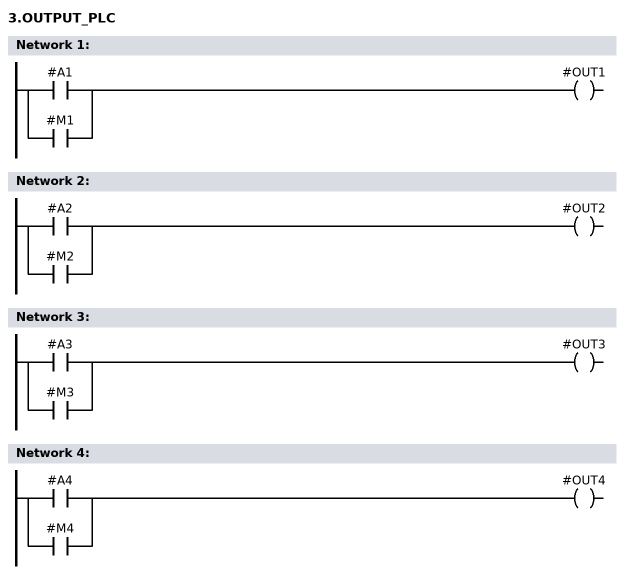
   RUNG wire#powerrail
      Contact( #A1 )
      wire#w1
      Coil( #OUT1 )
   END_RUNG
   RUNG wire#powerrail
      Contact( #M1 )
   END_RUNG wire#w1
   // the same network as SCL:
   #OUT1 := #A1 OR #M1;
END_REGION

REGION Network 2
   RUNG wire#powerrail
      Contact( #A2 )
      wire#w1
      Coil( #OUT2 )
   END_RUNG
   RUNG wire#powerrail
      Contact( #M2 )
   END_RUNG wire#w1
   // the same network as SCL:
   #OUT2 := #A2 OR #M2;
END_REGION

REGION Network 3
   RUNG wire#powerrail
      Contact( #A3 )
      wire#w1
      Coil( #OUT3 )
   END_RUNG
   RUNG wire#powerrail
      Contact( #M3 )
   END_RUNG wire#w1
   // the same network as SCL:
   #OUT3 := #A3 OR #M3;
END_REGION

REGION Network 4
   RUNG wire#powerrail
      Contact( #A4 )
      wire#w1
      Coil( #OUT4 )
   END_RUNG
   RUNG wire#powerrail
      Contact( #M4 )
   END_RUNG wire#w1
   // the same network as SCL:
   #OUT4 := #A4 OR #M4;
END_REGION
END_FUNCTION

FUNCTION_BLOCK "3.RUN_MODE"   // FB3, LAD
{ S7_Optimized_Access := 'TRUE' }
VERSION : 0.1
// stored: AutoNumber false, CodeModifiedDate 2025-08-27T17:11:43.2955348Z, CompileDate 2026-01-15T16:25:55.5692242Z, CreationDate 2026-01-15T16:22:49.8270549Z, DownloadWithoutReinit false, HandleErrorsWithinBlock false, InterfaceModifiedDate 2023-07-24T14:42:19.3789304Z, IsConsistent true, IsIECCheckEnabled false, IsKnowHowProtected false, IsRetainMemResEnabled false, IsWriteProtected false, LibraryConformanceStatus The object is library-conformant., MemoryReserve 100, ModifiedDate 2025-08-27T17:11:43.2955348Z, ParameterModified 2023-07-24T14:41:56.9787559Z, PLCSimAdvancedSupport false, SetENOAutomatically False, StructureModified 2023-07-24T14:42:19.3789304Z, UDAEnableTagReadback false
   VAR_INPUT
      NN_RUN : Bool;
      NN_STOP : Bool;
      SW_SIM : Bool;
      SW_MAN : Bool;
      SW_AUT : Bool;
   END_VAR
   VAR_OUTPUT
      RUN : Bool;
      SIM : Bool;
      MAN : Bool;
      AUT : Bool;
   END_VAR
   VAR
      TEMP1 : Bool;
      TEMP2 : Bool;
   END_VAR
BEGIN

REGION Network 1
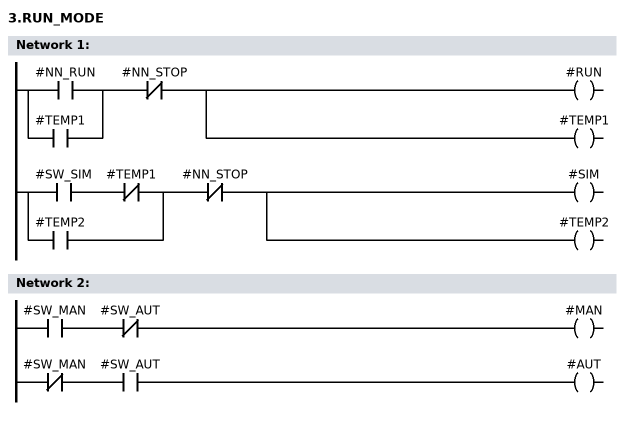
   RUNG wire#powerrail
      Contact( #NN_RUN )
      wire#w1
      I_Contact( #NN_STOP )
      wire#w2
      Coil( #RUN )
   END_RUNG
   RUNG wire#powerrail
      Contact( #TEMP1 )
   END_RUNG wire#w1
   RUNG wire#w2
      Coil( #TEMP1 )
   END_RUNG
   RUNG wire#powerrail
      Contact( #SW_SIM )
      I_Contact( #TEMP1 )
      wire#w3
      I_Contact( #NN_STOP )
      wire#w4
      Coil( #SIM )
   END_RUNG
   RUNG wire#powerrail
      Contact( #TEMP2 )
   END_RUNG wire#w3
   RUNG wire#w4
      Coil( #TEMP2 )
   END_RUNG
   // the same network as SCL:
   #RUN := (#NN_RUN OR #TEMP1) AND NOT #NN_STOP;
   #TEMP1 := #RUN;
   #SIM := ((#SW_SIM AND NOT #TEMP1) OR #TEMP2) AND NOT #NN_STOP;
   #TEMP2 := #SIM;
END_REGION

REGION Network 2
   RUNG wire#powerrail
      Contact( #SW_MAN )
      I_Contact( #SW_AUT )
      Coil( #MAN )
   END_RUNG
   RUNG wire#powerrail
      I_Contact( #SW_MAN )
      Contact( #SW_AUT )
      Coil( #AUT )
   END_RUNG
   // the same network as SCL:
   #MAN := #SW_MAN AND NOT #SW_AUT;
   #AUT := NOT #SW_MAN AND #SW_AUT;
END_REGION
END_FUNCTION_BLOCK

FUNCTION "4.CONVERT_VOLUME" : Void   // FC4, LAD
{ S7_Optimized_Access := 'TRUE' }
VERSION : 0.1
// stored: AutoNumber true, CodeModifiedDate 2025-08-27T17:08:03.467369Z, CompileDate 2026-01-15T16:25:55.7118746Z, CreationDate 2026-01-15T16:22:49.8270549Z, HandleErrorsWithinBlock false, InterfaceModifiedDate 2023-07-25T19:47:42.5745Z, IsConsistent true, IsIECCheckEnabled false, IsKnowHowProtected false, IsWriteProtected false, LibraryConformanceStatus The object is library-conformant., ModifiedDate 2025-08-27T17:08:03.467369Z, ParameterModified 2023-07-25T19:47:42.5745Z, PLCSimAdvancedSupport false, SetENOAutomatically False, StructureModified 2023-07-25T19:47:42.5745Z, UDAEnableTagReadback false
   VAR_INPUT
      SO_KHOI : Real;
      M3_MAX : Real;
   END_VAR
   VAR_OUTPUT
      SO_ME : Real;
      "M3/ME" : Real;
   END_VAR
   VAR_TEMP
      TEMP1 : Real;
      TEMP2 : Int;
      TEMP3 : Real;
   END_VAR
BEGIN

REGION Network 1
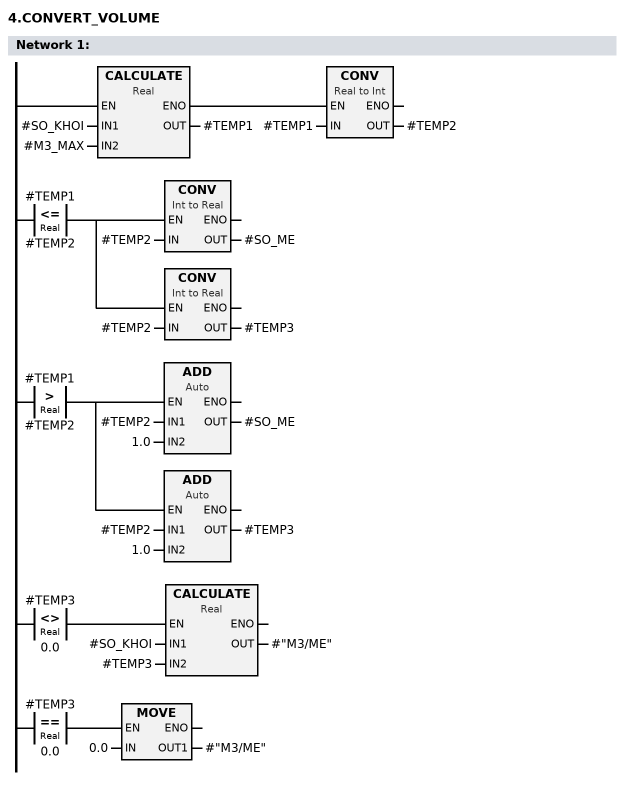
   RUNG wire#powerrail
      { S7_Templates := "SrcType := Real"; S7_Expression := "IN1/IN2" } Calculate(in1 := #SO_KHOI, in2 := #M3_MAX, out => #TEMP1)
      { S7_Templates := "[SrcType := Real, DestType := Int]" } Convert(in := #TEMP1, out => #TEMP2)
   END_RUNG
   RUNG wire#powerrail
      { S7_Templates := "SrcType := Real" } LE_Contact(in1 := #TEMP1, in2 := #TEMP2)
      wire#w1
      { S7_Templates := "[SrcType := Int, DestType := Real]" } Convert(in := #TEMP2, out => #SO_ME)
   END_RUNG
   RUNG wire#w1
      { S7_Templates := "[SrcType := Int, DestType := Real]" } Convert(in := #TEMP2, out => #TEMP3)
   END_RUNG
   RUNG wire#powerrail
      { S7_Templates := "SrcType := Real" } GT_Contact(in1 := #TEMP1, in2 := #TEMP2)
      wire#w2
      Add(in1 := #TEMP2, in2 := 1.0, out => #SO_ME)
   END_RUNG
   RUNG wire#w2
      Add(in1 := #TEMP2, in2 := 1.0, out => #TEMP3)
   END_RUNG
   RUNG wire#powerrail
      { S7_Templates := "SrcType := Real" } NE_Contact(in1 := #TEMP3, in2 := 0.0)
      { S7_Templates := "SrcType := Real"; S7_Expression := "IN1/IN2" } Calculate(in1 := #SO_KHOI, in2 := #TEMP3, out => #"M3/ME")
   END_RUNG
   RUNG wire#powerrail
      { S7_Templates := "SrcType := Real" } EQ_Contact(in1 := #TEMP3, in2 := 0.0)
      Move(in := 0.0, out1 => #"M3/ME")
   END_RUNG
   // the same network as SCL:
   #TEMP1 := #SO_KHOI/#M3_MAX;
   #TEMP2 := REAL_TO_INT(#TEMP1);
   IF #TEMP1 <= #TEMP2 THEN
       #SO_ME := INT_TO_REAL(#TEMP2);
       #TEMP3 := INT_TO_REAL(#TEMP2);
   END_IF;
   IF #TEMP1 > #TEMP2 THEN
       #SO_ME := #TEMP2 + 1.0;
       #TEMP3 := #TEMP2 + 1.0;
   END_IF;
   IF #TEMP3 <> 0.0 THEN #"M3/ME" := #SO_KHOI/#TEMP3; END_IF;
   IF #TEMP3 = 0.0 THEN #"M3/ME" := 0.0; END_IF;
END_REGION
END_FUNCTION

FUNCTION_BLOCK "5.ADDITIVES_PULE"   // FB5, LAD
{ S7_Optimized_Access := 'TRUE' }
VERSION : 0.1
// stored: AutoNumber false, CodeModifiedDate 2024-07-29T16:22:18.8856203Z, CompileDate 2026-01-15T16:25:55.5329987Z, CreationDate 2026-01-15T16:22:49.8270549Z, DownloadWithoutReinit false, HandleErrorsWithinBlock false, InterfaceModifiedDate 2024-07-29T16:20:48.5427985Z, IsConsistent true, IsIECCheckEnabled false, IsKnowHowProtected false, IsRetainMemResEnabled false, IsWriteProtected false, LibraryConformanceStatus The object is library-conformant., MemoryReserve 100, ModifiedDate 2024-07-29T16:22:18.8856203Z, ParameterModified 2024-07-29T16:20:48.5427985Z, PLCSimAdvancedSupport false, SetENOAutomatically False, StructureModified 2024-07-29T16:20:48.5427985Z, UDAEnableTagReadback false
   VAR_INPUT
      "Xung In" : DWord;
      Reset : Bool;
      "Set Tai" : Bool;
      "Khoi Luong Calib" : Real;
   END_VAR
   VAR_OUTPUT
      "Khoi Luong Out" : Real;
      "Xung Out" : Real;
   END_VAR
   VAR RETAIN
      "Xu In" : Real;
      "He So" : Real;
      "Xu Calib" : Real;
      "Kl Calib" : Real;
   END_VAR
   VAR
      M1 : Bool;
   END_VAR
   VAR_TEMP
      Conv : DInt;
   END_VAR
BEGIN

REGION Network 1
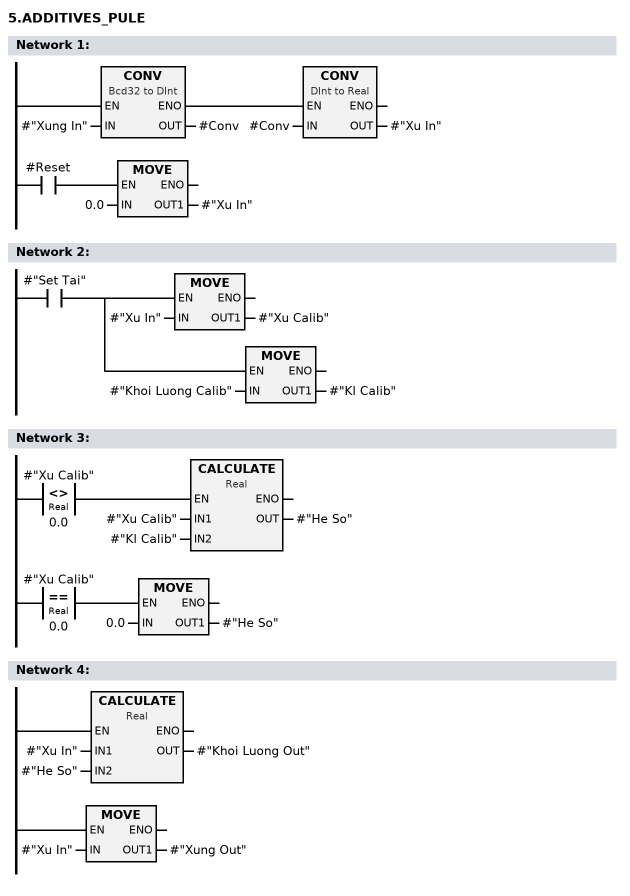
   RUNG wire#powerrail
      { S7_Templates := "[SrcType := Bcd32, DestType := DInt]" } Convert(in := #"Xung In", out => #Conv)
      { S7_Templates := "[SrcType := DInt, DestType := Real]" } Convert(in := #Conv, out => #"Xu In")
   END_RUNG
   RUNG wire#powerrail
      Contact( #Reset )
      Move(in := 0.0, out1 => #"Xu In")
   END_RUNG
   // the same network as SCL:
   #Conv := BCD32_TO_DINT(#"Xung In");
   #"Xu In" := DINT_TO_REAL(#Conv);
   IF #Reset THEN #"Xu In" := 0.0; END_IF;
END_REGION

REGION Network 2
   RUNG wire#powerrail
      Contact( #"Set Tai" )
      wire#w1
      Move(in := #"Xu In", out1 => #"Xu Calib")
   END_RUNG
   RUNG wire#w1
      Move(in := #"Khoi Luong Calib", out1 => #"Kl Calib")
   END_RUNG
   // the same network as SCL:
   IF #"Set Tai" THEN
       #"Xu Calib" := #"Xu In";
       #"Kl Calib" := #"Khoi Luong Calib";
   END_IF;
END_REGION

REGION Network 3
   RUNG wire#powerrail
      { S7_Templates := "SrcType := Real" } NE_Contact(in1 := #"Xu Calib", in2 := 0.0)
      { S7_Templates := "SrcType := Real"; S7_Expression := "IN2/IN1" } Calculate(in1 := #"Xu Calib", in2 := #"Kl Calib", out => #"He So")
   END_RUNG
   RUNG wire#powerrail
      { S7_Templates := "SrcType := Real" } EQ_Contact(in1 := #"Xu Calib", in2 := 0.0)
      Move(in := 0.0, out1 => #"He So")
   END_RUNG
   // the same network as SCL:
   IF #"Xu Calib" <> 0.0 THEN #"He So" := #"Kl Calib"/#"Xu Calib"; END_IF;
   IF #"Xu Calib" = 0.0 THEN #"He So" := 0.0; END_IF;
END_REGION

REGION Network 4
   RUNG wire#powerrail
      { S7_Templates := "SrcType := Real"; S7_Expression := "IN1*IN2" } Calculate(in1 := #"Xu In", in2 := #"He So", out => #"Khoi Luong Out")
   END_RUNG
   RUNG wire#powerrail
      Move(in := #"Xu In", out1 => #"Xung Out")
   END_RUNG
   // the same network as SCL:
   #"Khoi Luong Out" := #"Xu In"*#"He So";
   #"Xung Out" := #"Xu In";
END_REGION
END_FUNCTION_BLOCK

DATA_BLOCK "1.0 ANALOG_WAGG1"   // DB13
{ S7_Optimized_Access := 'TRUE' }
VERSION : 0.1
// stored: AutoNumber true, CodeModifiedDate 2026-01-15T16:25:52.6540779Z, CompileDate 2026-01-15T16:25:52.6593597Z, CreationDate 2026-01-15T16:22:49.8270549Z, DBAccessibleFromOPCUA true, DownloadWithoutReinit false, InstanceOfName 1.ANALOG_INPUT, InstanceOfNumber 1, InstanceOfType FB, InterfaceModifiedDate 2025-09-22T19:30:11.8403437Z, IsConsistent true, IsKnowHowProtected false, IsRetainMemResEnabled false, MemoryReserve 100, ModifiedDate 2026-01-15T16:25:52.6540779Z, ParameterModified 2025-08-30T17:31:01.4104373Z, StructureModified 2025-09-22T19:30:11.8403437Z, UDAEnableTagReadback false
"1.ANALOG_INPUT"
BEGIN
END_DATA_BLOCK

DATA_BLOCK "1.0 ANALOG_WAGG2"   // DB14
{ S7_Optimized_Access := 'TRUE' }
VERSION : 0.1
// stored: AutoNumber true, CodeModifiedDate 2026-01-15T16:25:52.3963656Z, CompileDate 2026-01-15T16:25:52.4020796Z, CreationDate 2026-01-15T16:22:49.8270549Z, DBAccessibleFromOPCUA true, DownloadWithoutReinit false, InstanceOfName 1.ANALOG_INPUT, InstanceOfNumber 1, InstanceOfType FB, InterfaceModifiedDate 2025-09-22T19:30:11.8403437Z, IsConsistent true, IsKnowHowProtected false, IsRetainMemResEnabled false, MemoryReserve 100, ModifiedDate 2026-01-15T16:25:52.3963656Z, ParameterModified 2025-08-30T17:31:01.4104373Z, StructureModified 2025-09-22T19:30:11.8403437Z, UDAEnableTagReadback false
"1.ANALOG_INPUT"
BEGIN
END_DATA_BLOCK

DATA_BLOCK "1.0 ANALOG_WAGG3"   // DB15
{ S7_Optimized_Access := 'TRUE' }
VERSION : 0.1
// stored: AutoNumber true, CodeModifiedDate 2026-01-15T16:25:52.7199099Z, CompileDate 2026-01-15T16:25:52.7268374Z, CreationDate 2026-01-15T16:22:49.8270549Z, DBAccessibleFromOPCUA true, DownloadWithoutReinit false, InstanceOfName 1.ANALOG_INPUT, InstanceOfNumber 1, InstanceOfType FB, InterfaceModifiedDate 2025-09-22T19:30:11.8403437Z, IsConsistent true, IsKnowHowProtected false, IsRetainMemResEnabled false, MemoryReserve 100, ModifiedDate 2026-01-15T16:25:52.7199099Z, ParameterModified 2025-08-30T17:31:01.4104373Z, StructureModified 2025-09-22T19:30:11.8403437Z, UDAEnableTagReadback false
"1.ANALOG_INPUT"
BEGIN
END_DATA_BLOCK

DATA_BLOCK "1.0 ANALOG_WAGG4"   // DB16
{ S7_Optimized_Access := 'TRUE' }
VERSION : 0.1
// stored: AutoNumber true, CodeModifiedDate 2026-01-15T16:25:52.7373182Z, CompileDate 2026-01-15T16:25:52.7414895Z, CreationDate 2026-01-15T16:22:49.8270549Z, DBAccessibleFromOPCUA true, DownloadWithoutReinit false, InstanceOfName 1.ANALOG_INPUT, InstanceOfNumber 1, InstanceOfType FB, InterfaceModifiedDate 2025-09-22T19:30:11.8403437Z, IsConsistent true, IsKnowHowProtected false, IsRetainMemResEnabled false, MemoryReserve 100, ModifiedDate 2026-01-15T16:25:52.7373182Z, ParameterModified 2025-08-30T17:31:01.4104373Z, StructureModified 2025-09-22T19:30:11.8403437Z, UDAEnableTagReadback false
"1.ANALOG_INPUT"
BEGIN
END_DATA_BLOCK

DATA_BLOCK "1.0 ANALOG_WAGG5"   // DB17
{ S7_Optimized_Access := 'TRUE' }
VERSION : 0.1
// stored: AutoNumber true, CodeModifiedDate 2026-01-15T16:25:52.7694615Z, CompileDate 2026-01-15T16:25:52.774821Z, CreationDate 2026-01-15T16:22:49.8270549Z, DBAccessibleFromOPCUA true, DownloadWithoutReinit false, InstanceOfName 1.ANALOG_INPUT, InstanceOfNumber 1, InstanceOfType FB, InterfaceModifiedDate 2025-09-22T19:30:11.8403437Z, IsConsistent true, IsKnowHowProtected false, IsRetainMemResEnabled false, MemoryReserve 100, ModifiedDate 2026-01-15T16:25:52.7694615Z, ParameterModified 2025-08-30T17:31:01.4104373Z, StructureModified 2025-09-22T19:30:11.8403437Z, UDAEnableTagReadback false
"1.ANALOG_INPUT"
BEGIN
END_DATA_BLOCK

DATA_BLOCK "1.0.ANALOG_WAG"   // DB100
{ S7_Optimized_Access := 'TRUE' }
VERSION : 0.1
// stored: AutoNumber false, CodeModifiedDate 2026-01-15T16:25:52.8141253Z, CompileDate 2026-01-15T16:25:52.8191872Z, CreationDate 2026-01-15T16:22:49.8270549Z, DBAccessibleFromOPCUA true, DownloadWithoutReinit false, InstanceOfName 1.ANALOG_INPUT, InstanceOfNumber 1, InstanceOfType FB, InterfaceModifiedDate 2025-09-22T19:30:11.8403437Z, IsConsistent true, IsKnowHowProtected false, IsRetainMemResEnabled false, MemoryReserve 100, ModifiedDate 2026-01-15T16:25:52.8141253Z, ParameterModified 2025-08-30T17:31:01.4104373Z, StructureModified 2025-09-22T19:30:11.8403437Z, UDAEnableTagReadback false
"1.ANALOG_INPUT"
BEGIN
END_DATA_BLOCK

DATA_BLOCK "1.0.ANALOG_WAP"   // DB102
{ S7_Optimized_Access := 'TRUE' }
VERSION : 0.1
// stored: AutoNumber false, CodeModifiedDate 2026-01-15T16:25:52.7536626Z, CompileDate 2026-01-15T16:25:52.7573094Z, CreationDate 2026-01-15T16:22:49.8270549Z, DBAccessibleFromOPCUA true, DownloadWithoutReinit false, InstanceOfName 1.ANALOG_INPUT, InstanceOfNumber 1, InstanceOfType FB, InterfaceModifiedDate 2025-09-22T19:30:11.8403437Z, IsConsistent true, IsKnowHowProtected false, IsRetainMemResEnabled false, MemoryReserve 100, ModifiedDate 2026-01-15T16:25:52.7536626Z, ParameterModified 2025-08-30T17:31:01.4104373Z, StructureModified 2025-09-22T19:30:11.8403437Z, UDAEnableTagReadback false
"1.ANALOG_INPUT"
BEGIN
END_DATA_BLOCK

DATA_BLOCK "1.0.ANALOG_WFD"   // DB101
{ S7_Optimized_Access := 'TRUE' }
VERSION : 0.1
// stored: AutoNumber false, CodeModifiedDate 2026-01-15T16:25:52.8468079Z, CompileDate 2026-01-15T16:25:52.8528873Z, CreationDate 2026-01-15T16:22:49.8270549Z, DBAccessibleFromOPCUA true, DownloadWithoutReinit false, InstanceOfName 1.ANALOG_INPUT, InstanceOfNumber 1, InstanceOfType FB, InterfaceModifiedDate 2025-09-22T19:30:11.8403437Z, IsConsistent true, IsKnowHowProtected false, IsRetainMemResEnabled false, MemoryReserve 100, ModifiedDate 2026-01-15T16:25:52.8468079Z, ParameterModified 2025-08-30T17:31:01.4104373Z, StructureModified 2025-09-22T19:30:11.8403437Z, UDAEnableTagReadback false
"1.ANALOG_INPUT"
BEGIN
END_DATA_BLOCK

DATA_BLOCK "1.0.ANALOG_WSBS"   // DB103
{ S7_Optimized_Access := 'TRUE' }
VERSION : 0.1
// stored: AutoNumber false, CodeModifiedDate 2026-01-15T16:25:52.4129937Z, CompileDate 2026-01-15T16:25:52.41757Z, CreationDate 2026-01-15T16:22:49.8270549Z, DBAccessibleFromOPCUA true, DownloadWithoutReinit false, InstanceOfName 1.ANALOG_INPUT, InstanceOfNumber 1, InstanceOfType FB, InterfaceModifiedDate 2025-09-22T19:30:11.8403437Z, IsConsistent true, IsKnowHowProtected false, IsRetainMemResEnabled false, MemoryReserve 100, ModifiedDate 2026-01-15T16:25:52.4129937Z, ParameterModified 2025-08-30T17:31:01.4104373Z, StructureModified 2025-09-22T19:30:11.8403437Z, UDAEnableTagReadback false
"1.ANALOG_INPUT"
BEGIN
END_DATA_BLOCK

DATA_BLOCK "1.1.ANALOG_TEMP_AG"   // DB107
{ S7_Optimized_Access := 'TRUE' }
VERSION : 0.1
// stored: AutoNumber false, CodeModifiedDate 2026-01-15T16:25:55.2427554Z, CompileDate 2026-01-15T16:25:55.2463904Z, CreationDate 2026-01-15T16:22:49.8270549Z, DBAccessibleFromOPCUA true, DownloadWithoutReinit false, InstanceOfName 1.ANALOG_INPUT, InstanceOfNumber 1, InstanceOfType FB, InterfaceModifiedDate 2025-09-22T19:30:11.8403437Z, IsConsistent true, IsKnowHowProtected false, IsRetainMemResEnabled false, MemoryReserve 100, ModifiedDate 2026-01-15T16:25:55.2427554Z, ParameterModified 2025-08-30T17:31:01.4104373Z, StructureModified 2025-09-22T19:30:11.8403437Z, UDAEnableTagReadback false
"1.ANALOG_INPUT"
BEGIN
END_DATA_BLOCK

DATA_BLOCK "1.1.ANALOG_TEMP_AP"   // DB106
{ S7_Optimized_Access := 'TRUE' }
VERSION : 0.1
// stored: AutoNumber false, CodeModifiedDate 2026-01-15T16:25:55.2265108Z, CompileDate 2026-01-15T16:25:55.2310383Z, CreationDate 2026-01-15T16:22:49.8270549Z, DBAccessibleFromOPCUA true, DownloadWithoutReinit false, InstanceOfName 1.ANALOG_INPUT, InstanceOfNumber 1, InstanceOfType FB, InterfaceModifiedDate 2025-09-22T19:30:11.8403437Z, IsConsistent true, IsKnowHowProtected false, IsRetainMemResEnabled false, MemoryReserve 100, ModifiedDate 2026-01-15T16:25:55.2265108Z, ParameterModified 2025-08-30T17:31:01.4104373Z, StructureModified 2025-09-22T19:30:11.8403437Z, UDAEnableTagReadback false
"1.ANALOG_INPUT"
BEGIN
END_DATA_BLOCK

DATA_BLOCK "1.1.ANALOG_TEMP_TL"   // DB104
{ S7_Optimized_Access := 'TRUE' }
VERSION : 0.1
// stored: AutoNumber false, CodeModifiedDate 2026-01-15T16:25:55.1844159Z, CompileDate 2026-01-15T16:25:55.1909886Z, CreationDate 2026-01-15T16:22:49.8270549Z, DBAccessibleFromOPCUA true, DownloadWithoutReinit false, InstanceOfName 1.ANALOG_INPUT, InstanceOfNumber 1, InstanceOfType FB, InterfaceModifiedDate 2025-09-22T19:30:11.8403437Z, IsConsistent true, IsKnowHowProtected false, IsRetainMemResEnabled false, MemoryReserve 100, ModifiedDate 2026-01-15T16:25:55.1844159Z, ParameterModified 2025-08-30T17:31:01.4104373Z, StructureModified 2025-09-22T19:30:11.8403437Z, UDAEnableTagReadback false
"1.ANALOG_INPUT"
BEGIN
END_DATA_BLOCK

DATA_BLOCK "1.1.ANALOG_TEMP_TS"   // DB105
{ S7_Optimized_Access := 'TRUE' }
VERSION : 0.1
// stored: AutoNumber false, CodeModifiedDate 2026-01-15T16:25:55.2062711Z, CompileDate 2026-01-15T16:25:55.2133319Z, CreationDate 2026-01-15T16:22:49.8270549Z, DBAccessibleFromOPCUA true, DownloadWithoutReinit false, InstanceOfName 1.ANALOG_INPUT, InstanceOfNumber 1, InstanceOfType FB, InterfaceModifiedDate 2025-09-22T19:30:11.8403437Z, IsConsistent true, IsKnowHowProtected false, IsRetainMemResEnabled false, MemoryReserve 100, ModifiedDate 2026-01-15T16:25:55.2062711Z, ParameterModified 2025-08-30T17:31:01.4104373Z, StructureModified 2025-09-22T19:30:11.8403437Z, UDAEnableTagReadback false
"1.ANALOG_INPUT"
BEGIN
END_DATA_BLOCK

DATA_BLOCK "10.0.RUNG_AGG1"   // DB1000
{ S7_Optimized_Access := 'TRUE' }
VERSION : 0.1
// stored: AutoNumber false, CodeModifiedDate 2026-01-15T16:25:55.7954208Z, CompileDate 2026-01-15T16:25:55.801975Z, CreationDate 2026-01-15T16:22:49.8270549Z, DBAccessibleFromOPCUA true, DownloadWithoutReinit false, InstanceOfName 10.TIMER_CLOCK, InstanceOfNumber 10, InstanceOfType FB, InterfaceModifiedDate 2023-08-14T08:08:19.3737097Z, IsConsistent true, IsKnowHowProtected false, IsRetainMemResEnabled false, MemoryReserve 100, ModifiedDate 2026-01-15T16:25:55.7954208Z, ParameterModified 2022-05-24T16:04:05.0982286Z, StructureModified 2023-08-14T08:08:19.3737097Z, UDAEnableTagReadback false
"10.TIMER_CLOCK"
BEGIN
END_DATA_BLOCK

DATA_BLOCK "10.1.RUNG_CE1"   // DB1006
{ S7_Optimized_Access := 'TRUE' }
VERSION : 0.1
// stored: AutoNumber false, CodeModifiedDate 2026-01-15T16:25:55.7775419Z, CompileDate 2026-01-15T16:25:55.7820883Z, CreationDate 2026-01-15T16:22:49.8270549Z, DBAccessibleFromOPCUA true, DownloadWithoutReinit false, InstanceOfName 10.TIMER_CLOCK, InstanceOfNumber 10, InstanceOfType FB, InterfaceModifiedDate 2023-08-14T08:08:19.3737097Z, IsConsistent true, IsKnowHowProtected false, IsRetainMemResEnabled false, MemoryReserve 100, ModifiedDate 2026-01-15T16:25:55.7775419Z, ParameterModified 2022-05-24T16:04:05.0982286Z, StructureModified 2023-08-14T08:08:19.3737097Z, UDAEnableTagReadback false
"10.TIMER_CLOCK"
BEGIN
END_DATA_BLOCK

DATA_BLOCK "10.3.SKSL_1"   // DB1009
{ S7_Optimized_Access := 'TRUE' }
VERSION : 0.1
// stored: AutoNumber false, CodeModifiedDate 2026-01-15T16:25:55.7623037Z, CompileDate 2026-01-15T16:25:55.7683704Z, CreationDate 2026-01-15T16:22:49.8270549Z, DBAccessibleFromOPCUA true, DownloadWithoutReinit false, InstanceOfName 10.TIMER_CLOCK, InstanceOfNumber 10, InstanceOfType FB, InterfaceModifiedDate 2023-08-14T08:08:19.3737097Z, IsConsistent true, IsKnowHowProtected false, IsRetainMemResEnabled false, MemoryReserve 100, ModifiedDate 2026-01-15T16:25:55.7623037Z, ParameterModified 2022-05-24T16:04:05.0982286Z, StructureModified 2023-08-14T08:08:19.3737097Z, UDAEnableTagReadback false
"10.TIMER_CLOCK"
BEGIN
END_DATA_BLOCK

DATA_BLOCK "2.0_NN0_0"   // DB200
{ S7_Optimized_Access := 'TRUE' }
VERSION : 0.1
// stored: AutoNumber false, CodeModifiedDate 2025-08-27T17:14:33.7093845Z, CompileDate 2026-01-15T16:25:52.803973Z, CreationDate 2026-01-15T16:22:49.8270549Z, DBAccessibleFromOPCUA true, DownloadWithoutReinit false, InstanceOfName 2.MANUAL_CONTROL, InstanceOfNumber 2, InstanceOfType FB, InterfaceModifiedDate 2025-08-27T17:14:33.2091456Z, IsConsistent true, IsKnowHowProtected false, IsRetainMemResEnabled false, MemoryReserve 100, ModifiedDate 2025-08-27T17:14:33.7093845Z, ParameterModified 2024-10-13T14:59:19.5830719Z, StructureModified 2025-08-27T17:14:33.2091456Z, UDAEnableTagReadback false
"2.MANUAL_CONTROL"
BEGIN
END_DATA_BLOCK

DATA_BLOCK "2.0_NN0_1"   // DB201
{ S7_Optimized_Access := 'TRUE' }
VERSION : 0.1
// stored: AutoNumber false, CodeModifiedDate 2025-08-27T17:14:33.6624193Z, CompileDate 2026-01-15T16:25:52.6174369Z, CreationDate 2026-01-15T16:22:49.8270549Z, DBAccessibleFromOPCUA true, DownloadWithoutReinit false, InstanceOfName 2.MANUAL_CONTROL, InstanceOfNumber 2, InstanceOfType FB, InterfaceModifiedDate 2025-08-27T17:14:33.2091456Z, IsConsistent true, IsKnowHowProtected false, IsRetainMemResEnabled false, MemoryReserve 100, ModifiedDate 2025-08-27T17:14:33.6624193Z, ParameterModified 2024-10-13T14:59:19.5830719Z, StructureModified 2025-08-27T17:14:33.2091456Z, UDAEnableTagReadback false
"2.MANUAL_CONTROL"
BEGIN
END_DATA_BLOCK

DATA_BLOCK "2.0_NN0_2"   // DB202
{ S7_Optimized_Access := 'TRUE' }
VERSION : 0.1
// stored: AutoNumber false, CodeModifiedDate 2025-08-27T17:14:33.8028627Z, CompileDate 2026-01-15T16:25:52.6287047Z, CreationDate 2026-01-15T16:22:49.8270549Z, DBAccessibleFromOPCUA true, DownloadWithoutReinit false, InstanceOfName 2.MANUAL_CONTROL, InstanceOfNumber 2, InstanceOfType FB, InterfaceModifiedDate 2025-08-27T17:14:33.2091456Z, IsConsistent true, IsKnowHowProtected false, IsRetainMemResEnabled false, MemoryReserve 100, ModifiedDate 2025-08-27T17:14:33.8028627Z, ParameterModified 2024-10-13T14:59:19.5830719Z, StructureModified 2025-08-27T17:14:33.2091456Z, UDAEnableTagReadback false
"2.MANUAL_CONTROL"
BEGIN
END_DATA_BLOCK

DATA_BLOCK "2.0_NN0_3"   // DB203
{ S7_Optimized_Access := 'TRUE' }
VERSION : 0.1
// stored: AutoNumber false, CodeModifiedDate 2025-08-27T17:14:33.7717804Z, CompileDate 2026-01-15T16:25:52.6419409Z, CreationDate 2026-01-15T16:22:49.8270549Z, DBAccessibleFromOPCUA true, DownloadWithoutReinit false, InstanceOfName 2.MANUAL_CONTROL, InstanceOfNumber 2, InstanceOfType FB, InterfaceModifiedDate 2025-08-27T17:14:33.2091456Z, IsConsistent true, IsKnowHowProtected false, IsRetainMemResEnabled false, MemoryReserve 100, ModifiedDate 2025-08-27T17:14:33.7717804Z, ParameterModified 2024-10-13T14:59:19.5830719Z, StructureModified 2025-08-27T17:14:33.2091456Z, UDAEnableTagReadback false
"2.MANUAL_CONTROL"
BEGIN
END_DATA_BLOCK

DATA_BLOCK "2.0_NN0_4"   // DB204
{ S7_Optimized_Access := 'TRUE' }
VERSION : 0.1
// stored: AutoNumber false, CodeModifiedDate 2025-08-27T17:14:33.7717798Z, CompileDate 2026-01-15T16:25:55.1732612Z, CreationDate 2026-01-15T16:22:49.8270549Z, DBAccessibleFromOPCUA true, DownloadWithoutReinit false, InstanceOfName 2.MANUAL_CONTROL, InstanceOfNumber 2, InstanceOfType FB, InterfaceModifiedDate 2025-08-27T17:14:33.2091456Z, IsConsistent true, IsKnowHowProtected false, IsRetainMemResEnabled false, MemoryReserve 100, ModifiedDate 2025-08-27T17:14:33.7717798Z, ParameterModified 2024-10-13T14:59:19.5830719Z, StructureModified 2025-08-27T17:14:33.2091456Z, UDAEnableTagReadback false
"2.MANUAL_CONTROL"
BEGIN
END_DATA_BLOCK

DATA_BLOCK "4.SIMULATION"   // DB400
{ S7_Optimized_Access := 'TRUE' }
VERSION : 0.1
// stored: AutoNumber false, CodeModifiedDate 2026-01-15T16:25:55.15091Z, CompileDate 2026-01-15T16:25:55.1580097Z, CreationDate 2026-01-15T16:22:49.8270549Z, DBAccessibleFromOPCUA true, DownloadWithoutReinit false, InstanceOfName 4.SIMULATION_DATA, InstanceOfNumber 4, InstanceOfType FB, InterfaceModifiedDate 2023-11-28T22:28:44.2264332Z, IsConsistent true, IsKnowHowProtected false, IsRetainMemResEnabled false, MemoryReserve 100, ModifiedDate 2026-01-15T16:25:55.15091Z, ParameterModified 2023-11-28T22:28:44.2264332Z, StructureModified 2023-11-28T22:28:44.2264332Z, UDAEnableTagReadback false
"4.SIMULATION_DATA"
BEGIN
END_DATA_BLOCK

DATA_BLOCK "6.1.WAGG1"   // DB601
{ S7_Optimized_Access := 'TRUE' }
VERSION : 0.1
// stored: AutoNumber false, CodeModifiedDate 2026-01-15T16:25:50.9109215Z, CompileDate 2026-01-15T16:25:50.9192936Z, CreationDate 2026-01-15T16:22:49.8270549Z, DBAccessibleFromOPCUA true, DownloadWithoutReinit false, InstanceOfName 6.WEIGHT_HANDLING, InstanceOfNumber 6, InstanceOfType FB, InterfaceModifiedDate 2023-12-29T17:39:18.5236469Z, IsConsistent true, IsKnowHowProtected false, IsRetainMemResEnabled false, MemoryReserve 100, ModifiedDate 2026-01-15T16:25:50.9109215Z, ParameterModified 2023-11-29T03:49:57.2782849Z, StructureModified 2023-12-29T17:39:18.5236469Z, UDAEnableTagReadback false
"6.WEIGHT_HANDLING"
BEGIN
END_DATA_BLOCK

DATA_BLOCK "6.1.W_IND_AGG1"   // DB19
{ S7_Optimized_Access := 'TRUE' }
VERSION : 0.1
// stored: AutoNumber true, CodeModifiedDate 2026-01-15T16:25:51.4257568Z, CompileDate 2026-01-15T16:25:51.429501Z, CreationDate 2026-01-15T16:22:49.8270549Z, DBAccessibleFromOPCUA true, DownloadWithoutReinit false, InstanceOfName 6.WEIGHT_HANDLING, InstanceOfNumber 6, InstanceOfType FB, InterfaceModifiedDate 2023-12-29T17:39:18.5236469Z, IsConsistent true, IsKnowHowProtected false, IsRetainMemResEnabled false, MemoryReserve 100, ModifiedDate 2026-01-15T16:25:51.4257568Z, ParameterModified 2023-11-29T03:49:57.2782849Z, StructureModified 2023-12-29T17:39:18.5236469Z, UDAEnableTagReadback false
"6.WEIGHT_HANDLING"
BEGIN
END_DATA_BLOCK

DATA_BLOCK "6.1.W_IND_AGG2"   // DB23
{ S7_Optimized_Access := 'TRUE' }
VERSION : 0.1
// stored: AutoNumber true, CodeModifiedDate 2026-01-15T16:25:52.0981926Z, CompileDate 2026-01-15T16:25:52.1042687Z, CreationDate 2026-01-15T16:22:49.8270549Z, DBAccessibleFromOPCUA true, DownloadWithoutReinit false, InstanceOfName 6.WEIGHT_HANDLING, InstanceOfNumber 6, InstanceOfType FB, InterfaceModifiedDate 2023-12-29T17:39:18.5236469Z, IsConsistent true, IsKnowHowProtected false, IsRetainMemResEnabled false, MemoryReserve 100, ModifiedDate 2026-01-15T16:25:52.0981926Z, ParameterModified 2023-11-29T03:49:57.2782849Z, StructureModified 2023-12-29T17:39:18.5236469Z, UDAEnableTagReadback false
"6.WEIGHT_HANDLING"
BEGIN
END_DATA_BLOCK

DATA_BLOCK "6.1.W_IND_AGG3"   // DB25
{ S7_Optimized_Access := 'TRUE' }
VERSION : 0.1
// stored: AutoNumber true, CodeModifiedDate 2026-01-15T16:25:52.1743928Z, CompileDate 2026-01-15T16:25:52.1820403Z, CreationDate 2026-01-15T16:22:49.8270549Z, DBAccessibleFromOPCUA true, DownloadWithoutReinit false, InstanceOfName 6.WEIGHT_HANDLING, InstanceOfNumber 6, InstanceOfType FB, InterfaceModifiedDate 2023-12-29T17:39:18.5236469Z, IsConsistent true, IsKnowHowProtected false, IsRetainMemResEnabled false, MemoryReserve 100, ModifiedDate 2026-01-15T16:25:52.1743928Z, ParameterModified 2023-11-29T03:49:57.2782849Z, StructureModified 2023-12-29T17:39:18.5236469Z, UDAEnableTagReadback false
"6.WEIGHT_HANDLING"
BEGIN
END_DATA_BLOCK

DATA_BLOCK "6.1.W_IND_AGG4"   // DB29
{ S7_Optimized_Access := 'TRUE' }
VERSION : 0.1
// stored: AutoNumber true, CodeModifiedDate 2026-01-15T16:25:52.0443037Z, CompileDate 2026-01-15T16:25:52.0495722Z, CreationDate 2026-01-15T16:22:49.8270549Z, DBAccessibleFromOPCUA true, DownloadWithoutReinit false, InstanceOfName 6.WEIGHT_HANDLING, InstanceOfNumber 6, InstanceOfType FB, InterfaceModifiedDate 2023-12-29T17:39:18.5236469Z, IsConsistent true, IsKnowHowProtected false, IsRetainMemResEnabled false, MemoryReserve 100, ModifiedDate 2026-01-15T16:25:52.0443037Z, ParameterModified 2023-11-29T03:49:57.2782849Z, StructureModified 2023-12-29T17:39:18.5236469Z, UDAEnableTagReadback false
"6.WEIGHT_HANDLING"
BEGIN
END_DATA_BLOCK

DATA_BLOCK "6.1.W_IND_AGG5"   // DB33
{ S7_Optimized_Access := 'TRUE' }
VERSION : 0.1
// stored: AutoNumber true, CodeModifiedDate 2026-01-15T16:25:51.9306777Z, CompileDate 2026-01-15T16:25:51.9357275Z, CreationDate 2026-01-15T16:22:49.8270549Z, DBAccessibleFromOPCUA true, DownloadWithoutReinit false, InstanceOfName 6.WEIGHT_HANDLING, InstanceOfNumber 6, InstanceOfType FB, InterfaceModifiedDate 2023-12-29T17:39:18.5236469Z, IsConsistent true, IsKnowHowProtected false, IsRetainMemResEnabled false, MemoryReserve 100, ModifiedDate 2026-01-15T16:25:51.9306777Z, ParameterModified 2023-11-29T03:49:57.2782849Z, StructureModified 2023-12-29T17:39:18.5236469Z, UDAEnableTagReadback false
"6.WEIGHT_HANDLING"
BEGIN
END_DATA_BLOCK

DATA_BLOCK "6.2.WCEM1"   // DB607
{ S7_Optimized_Access := 'TRUE' }
VERSION : 0.1
// stored: AutoNumber false, CodeModifiedDate 2026-01-15T16:25:51.2384683Z, CompileDate 2026-01-15T16:25:51.2440029Z, CreationDate 2026-01-15T16:22:49.8270549Z, DBAccessibleFromOPCUA true, DownloadWithoutReinit false, InstanceOfName 6.WEIGHT_HANDLING, InstanceOfNumber 6, InstanceOfType FB, InterfaceModifiedDate 2023-12-29T17:39:18.5236469Z, IsConsistent true, IsKnowHowProtected false, IsRetainMemResEnabled false, MemoryReserve 100, ModifiedDate 2026-01-15T16:25:51.2384683Z, ParameterModified 2023-11-29T03:49:57.2782849Z, StructureModified 2023-12-29T17:39:18.5236469Z, UDAEnableTagReadback false
"6.WEIGHT_HANDLING"
BEGIN
END_DATA_BLOCK

DATA_BLOCK "6.3.WWAT1"   // DB609
{ S7_Optimized_Access := 'TRUE' }
VERSION : 0.1
// stored: AutoNumber false, CodeModifiedDate 2026-01-15T16:25:51.1061526Z, CompileDate 2026-01-15T16:25:51.1117172Z, CreationDate 2026-01-15T16:22:49.8270549Z, DBAccessibleFromOPCUA true, DownloadWithoutReinit false, InstanceOfName 6.WEIGHT_HANDLING, InstanceOfNumber 6, InstanceOfType FB, InterfaceModifiedDate 2023-12-29T17:39:18.5236469Z, IsConsistent true, IsKnowHowProtected false, IsRetainMemResEnabled false, MemoryReserve 100, ModifiedDate 2026-01-15T16:25:51.1061526Z, ParameterModified 2023-11-29T03:49:57.2782849Z, StructureModified 2023-12-29T17:39:18.5236469Z, UDAEnableTagReadback false
"6.WEIGHT_HANDLING"
BEGIN
END_DATA_BLOCK

DATA_BLOCK "6.4.WADD1"   // DB611
{ S7_Optimized_Access := 'TRUE' }
VERSION : 0.1
// stored: AutoNumber false, CodeModifiedDate 2026-01-15T16:25:50.9806792Z, CompileDate 2026-01-15T16:25:50.9857091Z, CreationDate 2026-01-15T16:22:49.8270549Z, DBAccessibleFromOPCUA true, DownloadWithoutReinit false, InstanceOfName 6.WEIGHT_HANDLING, InstanceOfNumber 6, InstanceOfType FB, InterfaceModifiedDate 2023-12-29T17:39:18.5236469Z, IsConsistent true, IsKnowHowProtected false, IsRetainMemResEnabled false, MemoryReserve 100, ModifiedDate 2026-01-15T16:25:50.9806792Z, ParameterModified 2023-11-29T03:49:57.2782849Z, StructureModified 2023-12-29T17:39:18.5236469Z, UDAEnableTagReadback false
"6.WEIGHT_HANDLING"
BEGIN
END_DATA_BLOCK

DATA_BLOCK "7.1.AGG1"   // DB701
{ S7_Optimized_Access := 'TRUE' }
VERSION : 0.1
// stored: AutoNumber false, CodeModifiedDate 2026-01-15T16:25:50.9474767Z, CompileDate 2026-01-15T16:25:50.9530222Z, CreationDate 2026-01-15T16:22:49.8270549Z, DBAccessibleFromOPCUA true, DownloadWithoutReinit false, InstanceOfName 7.WEIGHT_PROCESS, InstanceOfNumber 7, InstanceOfType FB, InterfaceModifiedDate 2024-08-06T09:13:34.3012657Z, IsConsistent true, IsKnowHowProtected false, IsRetainMemResEnabled false, MemoryReserve 100, ModifiedDate 2026-01-15T16:25:50.9474767Z, ParameterModified 2024-08-06T08:53:48.4792275Z, StructureModified 2024-08-06T09:13:34.3012657Z, UDAEnableTagReadback false
"7.WEIGHT_PROCESS"
BEGIN
END_DATA_BLOCK

DATA_BLOCK "7.1.AGG2"   // DB702
{ S7_Optimized_Access := 'TRUE' }
VERSION : 0.1
// stored: AutoNumber false, CodeModifiedDate 2026-01-15T16:25:50.9657336Z, CompileDate 2026-01-15T16:25:50.9692801Z, CreationDate 2026-01-15T16:22:49.8270549Z, DBAccessibleFromOPCUA true, DownloadWithoutReinit false, InstanceOfName 7.WEIGHT_PROCESS, InstanceOfNumber 7, InstanceOfType FB, InterfaceModifiedDate 2024-08-06T09:13:34.3012657Z, IsConsistent true, IsKnowHowProtected false, IsRetainMemResEnabled false, MemoryReserve 100, ModifiedDate 2026-01-15T16:25:50.9657336Z, ParameterModified 2024-08-06T08:53:48.4792275Z, StructureModified 2024-08-06T09:13:34.3012657Z, UDAEnableTagReadback false
"7.WEIGHT_PROCESS"
BEGIN
END_DATA_BLOCK

DATA_BLOCK "7.1.AGG3"   // DB703
{ S7_Optimized_Access := 'TRUE' }
VERSION : 0.1
// stored: AutoNumber false, CodeModifiedDate 2026-01-15T16:25:51.0179497Z, CompileDate 2026-01-15T16:25:51.022606Z, CreationDate 2026-01-15T16:22:49.8270549Z, DBAccessibleFromOPCUA true, DownloadWithoutReinit false, InstanceOfName 7.WEIGHT_PROCESS, InstanceOfNumber 7, InstanceOfType FB, InterfaceModifiedDate 2024-08-06T09:13:34.3012657Z, IsConsistent true, IsKnowHowProtected false, IsRetainMemResEnabled false, MemoryReserve 100, ModifiedDate 2026-01-15T16:25:51.0179497Z, ParameterModified 2024-08-06T08:53:48.4792275Z, StructureModified 2024-08-06T09:13:34.3012657Z, UDAEnableTagReadback false
"7.WEIGHT_PROCESS"
BEGIN
END_DATA_BLOCK

DATA_BLOCK "7.1.AGG4"   // DB704
{ S7_Optimized_Access := 'TRUE' }
VERSION : 0.1
// stored: AutoNumber false, CodeModifiedDate 2026-01-15T16:25:51.0501858Z, CompileDate 2026-01-15T16:25:51.0579472Z, CreationDate 2026-01-15T16:22:49.8270549Z, DBAccessibleFromOPCUA true, DownloadWithoutReinit false, InstanceOfName 7.WEIGHT_PROCESS, InstanceOfNumber 7, InstanceOfType FB, InterfaceModifiedDate 2024-08-06T09:13:34.3012657Z, IsConsistent true, IsKnowHowProtected false, IsRetainMemResEnabled false, MemoryReserve 100, ModifiedDate 2026-01-15T16:25:51.0501858Z, ParameterModified 2024-08-06T08:53:48.4792275Z, StructureModified 2024-08-06T09:13:34.3012657Z, UDAEnableTagReadback false
"7.WEIGHT_PROCESS"
BEGIN
END_DATA_BLOCK

DATA_BLOCK "7.1.AGG5"   // DB705
{ S7_Optimized_Access := 'TRUE' }
VERSION : 0.1
// stored: AutoNumber false, CodeModifiedDate 2026-01-15T16:25:51.3893687Z, CompileDate 2026-01-15T16:25:51.396597Z, CreationDate 2026-01-15T16:22:49.8270549Z, DBAccessibleFromOPCUA true, DownloadWithoutReinit false, InstanceOfName 7.WEIGHT_PROCESS, InstanceOfNumber 7, InstanceOfType FB, InterfaceModifiedDate 2024-08-06T09:13:34.3012657Z, IsConsistent true, IsKnowHowProtected false, IsRetainMemResEnabled false, MemoryReserve 100, ModifiedDate 2026-01-15T16:25:51.3893687Z, ParameterModified 2024-08-06T08:53:48.4792275Z, StructureModified 2024-08-06T09:13:34.3012657Z, UDAEnableTagReadback false
"7.WEIGHT_PROCESS"
BEGIN
END_DATA_BLOCK

DATA_BLOCK "7.1.IND_AGG1"   // DB18
{ S7_Optimized_Access := 'TRUE' }
VERSION : 0.1
// stored: AutoNumber true, CodeModifiedDate 2026-01-15T16:25:52.372783Z, CompileDate 2026-01-15T16:25:52.3794201Z, CreationDate 2026-01-15T16:22:49.8270549Z, DBAccessibleFromOPCUA true, DownloadWithoutReinit false, InstanceOfName 7.WEIGHT_PROCESS, InstanceOfNumber 7, InstanceOfType FB, InterfaceModifiedDate 2024-08-06T09:13:34.3012657Z, IsConsistent true, IsKnowHowProtected false, IsRetainMemResEnabled false, MemoryReserve 100, ModifiedDate 2026-01-15T16:25:52.372783Z, ParameterModified 2024-08-06T08:53:48.4792275Z, StructureModified 2024-08-06T09:13:34.3012657Z, UDAEnableTagReadback false
"7.WEIGHT_PROCESS"
BEGIN
END_DATA_BLOCK

DATA_BLOCK "7.1.IND_AGG2"   // DB22
{ S7_Optimized_Access := 'TRUE' }
VERSION : 0.1
// stored: AutoNumber true, CodeModifiedDate 2026-01-15T16:25:52.2192426Z, CompileDate 2026-01-15T16:25:52.2239061Z, CreationDate 2026-01-15T16:22:49.8270549Z, DBAccessibleFromOPCUA true, DownloadWithoutReinit false, InstanceOfName 7.WEIGHT_PROCESS, InstanceOfNumber 7, InstanceOfType FB, InterfaceModifiedDate 2024-08-06T09:13:34.3012657Z, IsConsistent true, IsKnowHowProtected false, IsRetainMemResEnabled false, MemoryReserve 100, ModifiedDate 2026-01-15T16:25:52.2192426Z, ParameterModified 2024-08-06T08:53:48.4792275Z, StructureModified 2024-08-06T09:13:34.3012657Z, UDAEnableTagReadback false
"7.WEIGHT_PROCESS"
BEGIN
END_DATA_BLOCK

DATA_BLOCK "7.1.IND_AGG3"   // DB27
{ S7_Optimized_Access := 'TRUE' }
VERSION : 0.1
// stored: AutoNumber true, CodeModifiedDate 2026-01-15T16:25:52.0775696Z, CompileDate 2026-01-15T16:25:52.0841706Z, CreationDate 2026-01-15T16:22:49.8270549Z, DBAccessibleFromOPCUA true, DownloadWithoutReinit false, InstanceOfName 7.WEIGHT_PROCESS, InstanceOfNumber 7, InstanceOfType FB, InterfaceModifiedDate 2024-08-06T09:13:34.3012657Z, IsConsistent true, IsKnowHowProtected false, IsRetainMemResEnabled false, MemoryReserve 100, ModifiedDate 2026-01-15T16:25:52.0775696Z, ParameterModified 2024-08-06T08:53:48.4792275Z, StructureModified 2024-08-06T09:13:34.3012657Z, UDAEnableTagReadback false
"7.WEIGHT_PROCESS"
BEGIN
END_DATA_BLOCK

DATA_BLOCK "7.1.IND_AGG4"   // DB32
{ S7_Optimized_Access := 'TRUE' }
VERSION : 0.1
// stored: AutoNumber true, CodeModifiedDate 2026-01-15T16:25:52.1182917Z, CompileDate 2026-01-15T16:25:52.1243097Z, CreationDate 2026-01-15T16:22:49.8270549Z, DBAccessibleFromOPCUA true, DownloadWithoutReinit false, InstanceOfName 7.WEIGHT_PROCESS, InstanceOfNumber 7, InstanceOfType FB, InterfaceModifiedDate 2024-08-06T09:13:34.3012657Z, IsConsistent true, IsKnowHowProtected false, IsRetainMemResEnabled false, MemoryReserve 100, ModifiedDate 2026-01-15T16:25:52.1182917Z, ParameterModified 2024-08-06T08:53:48.4792275Z, StructureModified 2024-08-06T09:13:34.3012657Z, UDAEnableTagReadback false
"7.WEIGHT_PROCESS"
BEGIN
END_DATA_BLOCK

DATA_BLOCK "7.1.IND_AGG5"   // DB36
{ S7_Optimized_Access := 'TRUE' }
VERSION : 0.1
// stored: AutoNumber true, CodeModifiedDate 2026-01-15T16:25:52.0080123Z, CompileDate 2026-01-15T16:25:52.0131868Z, CreationDate 2026-01-15T16:22:49.8270549Z, DBAccessibleFromOPCUA true, DownloadWithoutReinit false, InstanceOfName 7.WEIGHT_PROCESS, InstanceOfNumber 7, InstanceOfType FB, InterfaceModifiedDate 2024-08-06T09:13:34.3012657Z, IsConsistent true, IsKnowHowProtected false, IsRetainMemResEnabled false, MemoryReserve 100, ModifiedDate 2026-01-15T16:25:52.0080123Z, ParameterModified 2024-08-06T08:53:48.4792275Z, StructureModified 2024-08-06T09:13:34.3012657Z, UDAEnableTagReadback false
"7.WEIGHT_PROCESS"
BEGIN
END_DATA_BLOCK

DATA_BLOCK "7.2.CE1"   // DB707
{ S7_Optimized_Access := 'TRUE' }
VERSION : 0.1
// stored: AutoNumber false, CodeModifiedDate 2026-01-15T16:25:50.7983554Z, CompileDate 2026-01-15T16:25:50.841758Z, CreationDate 2026-01-15T16:22:49.8270549Z, DBAccessibleFromOPCUA true, DownloadWithoutReinit false, InstanceOfName 7.WEIGHT_PROCESS, InstanceOfNumber 7, InstanceOfType FB, InterfaceModifiedDate 2024-08-06T09:13:34.3012657Z, IsConsistent true, IsKnowHowProtected false, IsRetainMemResEnabled false, MemoryReserve 100, ModifiedDate 2026-01-15T16:25:50.7983554Z, ParameterModified 2024-08-06T08:53:48.4792275Z, StructureModified 2024-08-06T09:13:34.3012657Z, UDAEnableTagReadback false
"7.WEIGHT_PROCESS"
BEGIN
END_DATA_BLOCK

DATA_BLOCK "7.3.WA1"   // DB712
{ S7_Optimized_Access := 'TRUE' }
VERSION : 0.1
// stored: AutoNumber false, CodeModifiedDate 2026-01-15T16:25:51.3687471Z, CompileDate 2026-01-15T16:25:51.3740828Z, CreationDate 2026-01-15T16:22:49.8270549Z, DBAccessibleFromOPCUA true, DownloadWithoutReinit false, InstanceOfName 7.WEIGHT_PROCESS, InstanceOfNumber 7, InstanceOfType FB, InterfaceModifiedDate 2024-08-06T09:13:34.3012657Z, IsConsistent true, IsKnowHowProtected false, IsRetainMemResEnabled false, MemoryReserve 100, ModifiedDate 2026-01-15T16:25:51.3687471Z, ParameterModified 2024-08-06T08:53:48.4792275Z, StructureModified 2024-08-06T09:13:34.3012657Z, UDAEnableTagReadback false
"7.WEIGHT_PROCESS"
BEGIN
END_DATA_BLOCK

DATA_BLOCK "7.4.ADD1"   // DB714
{ S7_Optimized_Access := 'TRUE' }
VERSION : 0.1
// stored: AutoNumber false, CodeModifiedDate 2026-01-15T16:25:50.880886Z, CompileDate 2026-01-15T16:25:50.8878267Z, CreationDate 2026-01-15T16:22:49.8270549Z, DBAccessibleFromOPCUA true, DownloadWithoutReinit false, InstanceOfName 7.WEIGHT_PROCESS, InstanceOfNumber 7, InstanceOfType FB, InterfaceModifiedDate 2024-08-06T09:13:34.3012657Z, IsConsistent true, IsKnowHowProtected false, IsRetainMemResEnabled false, MemoryReserve 100, ModifiedDate 2026-01-15T16:25:50.880886Z, ParameterModified 2024-08-06T08:53:48.4792275Z, StructureModified 2024-08-06T09:13:34.3012657Z, UDAEnableTagReadback false
"7.WEIGHT_PROCESS"
BEGIN
END_DATA_BLOCK

DATA_BLOCK "7.4.ADD2"   // DB715
{ S7_Optimized_Access := 'TRUE' }
VERSION : 0.1
// stored: AutoNumber true, CodeModifiedDate 2026-01-15T16:25:55.8171738Z, CompileDate 2026-01-15T16:25:55.8220055Z, CreationDate 2026-01-15T16:22:49.8270549Z, DBAccessibleFromOPCUA true, DownloadWithoutReinit false, InstanceOfName 7.WEIGHT_PROCESS, InstanceOfNumber 7, InstanceOfType FB, InterfaceModifiedDate 2024-08-06T09:13:34.3012657Z, IsConsistent true, IsKnowHowProtected false, IsRetainMemResEnabled false, MemoryReserve 100, ModifiedDate 2026-01-15T16:25:55.8171738Z, ParameterModified 2024-08-06T08:53:48.4792275Z, StructureModified 2024-08-06T09:13:34.3012657Z, UDAEnableTagReadback false
"7.WEIGHT_PROCESS"
BEGIN
END_DATA_BLOCK

DATA_BLOCK "7.4.ADD3"   // DB716
{ S7_Optimized_Access := 'TRUE' }
VERSION : 0.1
// stored: AutoNumber true, CodeModifiedDate 2026-01-15T16:25:55.4818033Z, CompileDate 2026-01-15T16:25:55.4875483Z, CreationDate 2026-01-15T16:22:49.8270549Z, DBAccessibleFromOPCUA true, DownloadWithoutReinit false, InstanceOfName 7.WEIGHT_PROCESS, InstanceOfNumber 7, InstanceOfType FB, InterfaceModifiedDate 2024-08-06T09:13:34.3012657Z, IsConsistent true, IsKnowHowProtected false, IsRetainMemResEnabled false, MemoryReserve 100, ModifiedDate 2026-01-15T16:25:55.4818033Z, ParameterModified 2024-08-06T08:53:48.4792275Z, StructureModified 2024-08-06T09:13:34.3012657Z, UDAEnableTagReadback false
"7.WEIGHT_PROCESS"
BEGIN
END_DATA_BLOCK

DATA_BLOCK "7.4.ADD4"   // DB717
{ S7_Optimized_Access := 'TRUE' }
VERSION : 0.1
// stored: AutoNumber true, CodeModifiedDate 2026-01-15T16:25:55.9772968Z, CompileDate 2026-01-15T16:25:55.9813329Z, CreationDate 2026-01-15T16:22:49.8270549Z, DBAccessibleFromOPCUA true, DownloadWithoutReinit false, InstanceOfName 7.WEIGHT_PROCESS, InstanceOfNumber 7, InstanceOfType FB, InterfaceModifiedDate 2024-08-06T09:13:34.3012657Z, IsConsistent true, IsKnowHowProtected false, IsRetainMemResEnabled false, MemoryReserve 100, ModifiedDate 2026-01-15T16:25:55.9772968Z, ParameterModified 2024-08-06T08:53:48.4792275Z, StructureModified 2024-08-06T09:13:34.3012657Z, UDAEnableTagReadback false
"7.WEIGHT_PROCESS"
BEGIN
END_DATA_BLOCK

DATA_BLOCK "7.4.ADD5"   // DB718
{ S7_Optimized_Access := 'TRUE' }
VERSION : 0.1
// stored: AutoNumber true, CodeModifiedDate 2026-01-15T16:25:55.9575787Z, CompileDate 2026-01-15T16:25:55.9634896Z, CreationDate 2026-01-15T16:22:49.8270549Z, DBAccessibleFromOPCUA true, DownloadWithoutReinit false, InstanceOfName 7.WEIGHT_PROCESS, InstanceOfNumber 7, InstanceOfType FB, InterfaceModifiedDate 2024-08-06T09:13:34.3012657Z, IsConsistent true, IsKnowHowProtected false, IsRetainMemResEnabled false, MemoryReserve 100, ModifiedDate 2026-01-15T16:25:55.9575787Z, ParameterModified 2024-08-06T08:53:48.4792275Z, StructureModified 2024-08-06T09:13:34.3012657Z, UDAEnableTagReadback false
"7.WEIGHT_PROCESS"
BEGIN
END_DATA_BLOCK

DATA_BLOCK "7.4.ADD6"   // DB719
{ S7_Optimized_Access := 'TRUE' }
VERSION : 0.1
// stored: AutoNumber true, CodeModifiedDate 2026-01-15T16:25:55.9362535Z, CompileDate 2026-01-15T16:25:55.9409287Z, CreationDate 2026-01-15T16:22:49.8270549Z, DBAccessibleFromOPCUA true, DownloadWithoutReinit false, InstanceOfName 7.WEIGHT_PROCESS, InstanceOfNumber 7, InstanceOfType FB, InterfaceModifiedDate 2024-08-06T09:13:34.3012657Z, IsConsistent true, IsKnowHowProtected false, IsRetainMemResEnabled false, MemoryReserve 100, ModifiedDate 2026-01-15T16:25:55.9362535Z, ParameterModified 2024-08-06T08:53:48.4792275Z, StructureModified 2024-08-06T09:13:34.3012657Z, UDAEnableTagReadback false
"7.WEIGHT_PROCESS"
BEGIN
END_DATA_BLOCK

DATA_BLOCK "9.1.DLC_AGG1"   // DB901
{ S7_Optimized_Access := 'TRUE' }
VERSION : 0.1
// stored: AutoNumber false, CodeModifiedDate 2026-01-15T16:25:50.9332093Z, CompileDate 2026-01-15T16:25:50.9377517Z, CreationDate 2026-01-15T16:22:49.8270549Z, DBAccessibleFromOPCUA true, DownloadWithoutReinit false, InstanceOfName 9.TIMER_DELAY, InstanceOfNumber 9, InstanceOfType FB, InterfaceModifiedDate 2022-05-24T16:36:11.1705081Z, IsConsistent true, IsKnowHowProtected false, IsRetainMemResEnabled false, MemoryReserve 100, ModifiedDate 2026-01-15T16:25:50.9332093Z, ParameterModified 2022-05-24T16:36:11.1705081Z, StructureModified 2022-05-24T16:36:11.1705081Z, UDAEnableTagReadback false
"9.TIMER_DELAY"
BEGIN
END_DATA_BLOCK

DATA_BLOCK "9.1.DLC_AGG2"   // DB902
{ S7_Optimized_Access := 'TRUE' }
VERSION : 0.1
// stored: AutoNumber false, CodeModifiedDate 2026-01-15T16:25:51.0711702Z, CompileDate 2026-01-15T16:25:51.0771226Z, CreationDate 2026-01-15T16:22:49.8270549Z, DBAccessibleFromOPCUA true, DownloadWithoutReinit false, InstanceOfName 9.TIMER_DELAY, InstanceOfNumber 9, InstanceOfType FB, InterfaceModifiedDate 2022-05-24T16:36:11.1705081Z, IsConsistent true, IsKnowHowProtected false, IsRetainMemResEnabled false, MemoryReserve 100, ModifiedDate 2026-01-15T16:25:51.0711702Z, ParameterModified 2022-05-24T16:36:11.1705081Z, StructureModified 2022-05-24T16:36:11.1705081Z, UDAEnableTagReadback false
"9.TIMER_DELAY"
BEGIN
END_DATA_BLOCK

DATA_BLOCK "9.1.DLC_AGG3"   // DB903
{ S7_Optimized_Access := 'TRUE' }
VERSION : 0.1
// stored: AutoNumber false, CodeModifiedDate 2026-01-15T16:25:50.9985443Z, CompileDate 2026-01-15T16:25:51.0044444Z, CreationDate 2026-01-15T16:22:49.8270549Z, DBAccessibleFromOPCUA true, DownloadWithoutReinit false, InstanceOfName 9.TIMER_DELAY, InstanceOfNumber 9, InstanceOfType FB, InterfaceModifiedDate 2022-05-24T16:36:11.1705081Z, IsConsistent true, IsKnowHowProtected false, IsRetainMemResEnabled false, MemoryReserve 100, ModifiedDate 2026-01-15T16:25:50.9985443Z, ParameterModified 2022-05-24T16:36:11.1705081Z, StructureModified 2022-05-24T16:36:11.1705081Z, UDAEnableTagReadback false
"9.TIMER_DELAY"
BEGIN
END_DATA_BLOCK

DATA_BLOCK "9.1.DLC_AGG4"   // DB904
{ S7_Optimized_Access := 'TRUE' }
VERSION : 0.1
// stored: AutoNumber false, CodeModifiedDate 2026-01-15T16:25:51.409636Z, CompileDate 2026-01-15T16:25:51.4146153Z, CreationDate 2026-01-15T16:22:49.8270549Z, DBAccessibleFromOPCUA true, DownloadWithoutReinit false, InstanceOfName 9.TIMER_DELAY, InstanceOfNumber 9, InstanceOfType FB, InterfaceModifiedDate 2022-05-24T16:36:11.1705081Z, IsConsistent true, IsKnowHowProtected false, IsRetainMemResEnabled false, MemoryReserve 100, ModifiedDate 2026-01-15T16:25:51.409636Z, ParameterModified 2022-05-24T16:36:11.1705081Z, StructureModified 2022-05-24T16:36:11.1705081Z, UDAEnableTagReadback false
"9.TIMER_DELAY"
BEGIN
END_DATA_BLOCK

DATA_BLOCK "9.1.DLC_AGG5"   // DB905
{ S7_Optimized_Access := 'TRUE' }
VERSION : 0.1
// stored: AutoNumber false, CodeModifiedDate 2026-01-15T16:25:51.1493744Z, CompileDate 2026-01-15T16:25:51.1554173Z, CreationDate 2026-01-15T16:22:49.8270549Z, DBAccessibleFromOPCUA true, DownloadWithoutReinit false, InstanceOfName 9.TIMER_DELAY, InstanceOfNumber 9, InstanceOfType FB, InterfaceModifiedDate 2022-05-24T16:36:11.1705081Z, IsConsistent true, IsKnowHowProtected false, IsRetainMemResEnabled false, MemoryReserve 100, ModifiedDate 2026-01-15T16:25:51.1493744Z, ParameterModified 2022-05-24T16:36:11.1705081Z, StructureModified 2022-05-24T16:36:11.1705081Z, UDAEnableTagReadback false
"9.TIMER_DELAY"
BEGIN
END_DATA_BLOCK

DATA_BLOCK "9.1.DLC_IND_AGG1"   // DB955
{ S7_Optimized_Access := 'TRUE' }
VERSION : 0.1
// stored: AutoNumber false, CodeModifiedDate 2026-01-15T16:25:52.3481914Z, CompileDate 2026-01-15T16:25:52.3557777Z, CreationDate 2026-01-15T16:22:49.8270549Z, DBAccessibleFromOPCUA true, DownloadWithoutReinit false, InstanceOfName 9.TIMER_DELAY, InstanceOfNumber 9, InstanceOfType FB, InterfaceModifiedDate 2022-05-24T16:36:11.1705081Z, IsConsistent true, IsKnowHowProtected false, IsRetainMemResEnabled false, MemoryReserve 100, ModifiedDate 2026-01-15T16:25:52.3481914Z, ParameterModified 2022-05-24T16:36:11.1705081Z, StructureModified 2022-05-24T16:36:11.1705081Z, UDAEnableTagReadback false
"9.TIMER_DELAY"
BEGIN
END_DATA_BLOCK

DATA_BLOCK "9.1.DLC_IND_AGG2"   // DB21
{ S7_Optimized_Access := 'TRUE' }
VERSION : 0.1
// stored: AutoNumber true, CodeModifiedDate 2026-01-15T16:25:51.3083868Z, CompileDate 2026-01-15T16:25:51.3114166Z, CreationDate 2026-01-15T16:22:49.8270549Z, DBAccessibleFromOPCUA true, DownloadWithoutReinit false, InstanceOfName 9.TIMER_DELAY, InstanceOfNumber 9, InstanceOfType FB, InterfaceModifiedDate 2022-05-24T16:36:11.1705081Z, IsConsistent true, IsKnowHowProtected false, IsRetainMemResEnabled false, MemoryReserve 100, ModifiedDate 2026-01-15T16:25:51.3083868Z, ParameterModified 2022-05-24T16:36:11.1705081Z, StructureModified 2022-05-24T16:36:11.1705081Z, UDAEnableTagReadback false
"9.TIMER_DELAY"
BEGIN
END_DATA_BLOCK

DATA_BLOCK "9.1.DLC_IND_AGG3"   // DB26
{ S7_Optimized_Access := 'TRUE' }
VERSION : 0.1
// stored: AutoNumber true, CodeModifiedDate 2026-01-15T16:25:51.2609627Z, CompileDate 2026-01-15T16:25:51.266563Z, CreationDate 2026-01-15T16:22:49.8270549Z, DBAccessibleFromOPCUA true, DownloadWithoutReinit false, InstanceOfName 9.TIMER_DELAY, InstanceOfNumber 9, InstanceOfType FB, InterfaceModifiedDate 2022-05-24T16:36:11.1705081Z, IsConsistent true, IsKnowHowProtected false, IsRetainMemResEnabled false, MemoryReserve 100, ModifiedDate 2026-01-15T16:25:51.2609627Z, ParameterModified 2022-05-24T16:36:11.1705081Z, StructureModified 2022-05-24T16:36:11.1705081Z, UDAEnableTagReadback false
"9.TIMER_DELAY"
BEGIN
END_DATA_BLOCK

DATA_BLOCK "9.1.DLC_IND_AGG4"   // DB31
{ S7_Optimized_Access := 'TRUE' }
VERSION : 0.1
// stored: AutoNumber true, CodeModifiedDate 2026-01-15T16:25:51.2046379Z, CompileDate 2026-01-15T16:25:51.2091535Z, CreationDate 2026-01-15T16:22:49.8270549Z, DBAccessibleFromOPCUA true, DownloadWithoutReinit false, InstanceOfName 9.TIMER_DELAY, InstanceOfNumber 9, InstanceOfType FB, InterfaceModifiedDate 2022-05-24T16:36:11.1705081Z, IsConsistent true, IsKnowHowProtected false, IsRetainMemResEnabled false, MemoryReserve 100, ModifiedDate 2026-01-15T16:25:51.2046379Z, ParameterModified 2022-05-24T16:36:11.1705081Z, StructureModified 2022-05-24T16:36:11.1705081Z, UDAEnableTagReadback false
"9.TIMER_DELAY"
BEGIN
END_DATA_BLOCK

DATA_BLOCK "9.1.DLC_IND_AGG5"   // DB35
{ S7_Optimized_Access := 'TRUE' }
VERSION : 0.1
// stored: AutoNumber true, CodeModifiedDate 2026-01-15T16:25:51.1863411Z, CompileDate 2026-01-15T16:25:51.1921076Z, CreationDate 2026-01-15T16:22:49.8270549Z, DBAccessibleFromOPCUA true, DownloadWithoutReinit false, InstanceOfName 9.TIMER_DELAY, InstanceOfNumber 9, InstanceOfType FB, InterfaceModifiedDate 2022-05-24T16:36:11.1705081Z, IsConsistent true, IsKnowHowProtected false, IsRetainMemResEnabled false, MemoryReserve 100, ModifiedDate 2026-01-15T16:25:51.1863411Z, ParameterModified 2022-05-24T16:36:11.1705081Z, StructureModified 2022-05-24T16:36:11.1705081Z, UDAEnableTagReadback false
"9.TIMER_DELAY"
BEGIN
END_DATA_BLOCK

DATA_BLOCK "9.10.DELAY_FD1_SAU_AGG"   // DB939
{ S7_Optimized_Access := 'TRUE' }
VERSION : 0.1
// stored: AutoNumber false, CodeModifiedDate 2026-01-15T16:25:52.0612037Z, CompileDate 2026-01-15T16:25:52.0664388Z, CreationDate 2026-01-15T16:22:49.8270549Z, DBAccessibleFromOPCUA true, DownloadWithoutReinit false, InstanceOfName 9.TIMER_DELAY, InstanceOfNumber 9, InstanceOfType FB, InterfaceModifiedDate 2022-05-24T16:36:11.1705081Z, IsConsistent true, IsKnowHowProtected false, IsRetainMemResEnabled false, MemoryReserve 100, ModifiedDate 2026-01-15T16:25:52.0612037Z, ParameterModified 2022-05-24T16:36:11.1705081Z, StructureModified 2022-05-24T16:36:11.1705081Z, UDAEnableTagReadback false
"9.TIMER_DELAY"
BEGIN
END_DATA_BLOCK

DATA_BLOCK "9.10.DELAY_SB1_SAU_AGG"   // DB940
{ S7_Optimized_Access := 'TRUE' }
VERSION : 0.1
// stored: AutoNumber false, CodeModifiedDate 2026-01-15T16:25:51.3243492Z, CompileDate 2026-01-15T16:25:51.3279576Z, CreationDate 2026-01-15T16:22:49.8270549Z, DBAccessibleFromOPCUA true, DownloadWithoutReinit false, InstanceOfName 9.TIMER_DELAY, InstanceOfNumber 9, InstanceOfType FB, InterfaceModifiedDate 2022-05-24T16:36:11.1705081Z, IsConsistent true, IsKnowHowProtected false, IsRetainMemResEnabled false, MemoryReserve 100, ModifiedDate 2026-01-15T16:25:51.3243492Z, ParameterModified 2022-05-24T16:36:11.1705081Z, StructureModified 2022-05-24T16:36:11.1705081Z, UDAEnableTagReadback false
"9.TIMER_DELAY"
BEGIN
END_DATA_BLOCK

DATA_BLOCK "9.10.DELAY_TAT_BOM TUOI NHUA"   // DB941
{ S7_Optimized_Access := 'TRUE' }
VERSION : 0.1
// stored: AutoNumber false, CodeModifiedDate 2026-01-15T16:25:52.6708235Z, CompileDate 2026-01-15T16:25:52.6761188Z, CreationDate 2026-01-15T16:22:49.8270549Z, DBAccessibleFromOPCUA true, DownloadWithoutReinit false, InstanceOfName 9.TIMER_DELAY, InstanceOfNumber 9, InstanceOfType FB, InterfaceModifiedDate 2022-05-24T16:36:11.1705081Z, IsConsistent true, IsKnowHowProtected false, IsRetainMemResEnabled false, MemoryReserve 100, ModifiedDate 2026-01-15T16:25:52.6708235Z, ParameterModified 2022-05-24T16:36:11.1705081Z, StructureModified 2022-05-24T16:36:11.1705081Z, UDAEnableTagReadback false
"9.TIMER_DELAY"
BEGIN
END_DATA_BLOCK

DATA_BLOCK "9.11.DELAY_AP1_SAU_AGG"   // DB942
{ S7_Optimized_Access := 'TRUE' }
VERSION : 0.1
// stored: AutoNumber false, CodeModifiedDate 2026-01-15T16:25:51.3511497Z, CompileDate 2026-01-15T16:25:51.3563805Z, CreationDate 2026-01-15T16:22:49.8270549Z, DBAccessibleFromOPCUA true, DownloadWithoutReinit false, InstanceOfName 9.TIMER_DELAY, InstanceOfNumber 9, InstanceOfType FB, InterfaceModifiedDate 2022-05-24T16:36:11.1705081Z, IsConsistent true, IsKnowHowProtected false, IsRetainMemResEnabled false, MemoryReserve 100, ModifiedDate 2026-01-15T16:25:51.3511497Z, ParameterModified 2022-05-24T16:36:11.1705081Z, StructureModified 2022-05-24T16:36:11.1705081Z, UDAEnableTagReadback false
"9.TIMER_DELAY"
BEGIN
END_DATA_BLOCK

DATA_BLOCK "9.11.THOI_GIAN_TRON"   // DB944
{ S7_Optimized_Access := 'TRUE' }
VERSION : 0.1
// stored: AutoNumber false, CodeModifiedDate 2026-01-15T16:25:52.7847255Z, CompileDate 2026-01-15T16:25:52.7892478Z, CreationDate 2026-01-15T16:22:49.8270549Z, DBAccessibleFromOPCUA true, DownloadWithoutReinit false, InstanceOfName 9.TIMER_DELAY, InstanceOfNumber 9, InstanceOfType FB, InterfaceModifiedDate 2022-05-24T16:36:11.1705081Z, IsConsistent true, IsKnowHowProtected false, IsRetainMemResEnabled false, MemoryReserve 100, ModifiedDate 2026-01-15T16:25:52.7847255Z, ParameterModified 2022-05-24T16:36:11.1705081Z, StructureModified 2022-05-24T16:36:11.1705081Z, UDAEnableTagReadback false
"9.TIMER_DELAY"
BEGIN
END_DATA_BLOCK

DATA_BLOCK "9.12.THOI_GIAN_XA"   // DB945
{ S7_Optimized_Access := 'TRUE' }
VERSION : 0.1
// stored: AutoNumber false, CodeModifiedDate 2026-01-15T16:25:52.8305484Z, CompileDate 2026-01-15T16:25:52.8361777Z, CreationDate 2026-01-15T16:22:49.8270549Z, DBAccessibleFromOPCUA true, DownloadWithoutReinit false, InstanceOfName 9.TIMER_DELAY, InstanceOfNumber 9, InstanceOfType FB, InterfaceModifiedDate 2022-05-24T16:36:11.1705081Z, IsConsistent true, IsKnowHowProtected false, IsRetainMemResEnabled false, MemoryReserve 100, ModifiedDate 2026-01-15T16:25:52.8305484Z, ParameterModified 2022-05-24T16:36:11.1705081Z, StructureModified 2022-05-24T16:36:11.1705081Z, UDAEnableTagReadback false
"9.TIMER_DELAY"
BEGIN
END_DATA_BLOCK

DATA_BLOCK "9.13_RESET_SAVE"   // DB949
{ S7_Optimized_Access := 'TRUE' }
VERSION : 0.1
// stored: AutoNumber false, CodeModifiedDate 2026-01-15T16:25:52.9009525Z, CompileDate 2026-01-15T16:25:52.9040647Z, CreationDate 2026-01-15T16:22:49.8270549Z, DBAccessibleFromOPCUA true, DownloadWithoutReinit false, InstanceOfName 9.TIMER_DELAY, InstanceOfNumber 9, InstanceOfType FB, InterfaceModifiedDate 2022-05-24T16:36:11.1705081Z, IsConsistent true, IsKnowHowProtected false, IsRetainMemResEnabled false, MemoryReserve 100, ModifiedDate 2026-01-15T16:25:52.9009525Z, ParameterModified 2022-05-24T16:36:11.1705081Z, StructureModified 2022-05-24T16:36:11.1705081Z, UDAEnableTagReadback false
"9.TIMER_DELAY"
BEGIN
END_DATA_BLOCK

DATA_BLOCK "9.2.DLC_CE1"   // DB907
{ S7_Optimized_Access := 'TRUE' }
VERSION : 0.1
// stored: AutoNumber false, CodeModifiedDate 2026-01-15T16:25:51.2232571Z, CompileDate 2026-01-15T16:25:51.2274478Z, CreationDate 2026-01-15T16:22:49.8270549Z, DBAccessibleFromOPCUA true, DownloadWithoutReinit false, InstanceOfName 9.TIMER_DELAY, InstanceOfNumber 9, InstanceOfType FB, InterfaceModifiedDate 2022-05-24T16:36:11.1705081Z, IsConsistent true, IsKnowHowProtected false, IsRetainMemResEnabled false, MemoryReserve 100, ModifiedDate 2026-01-15T16:25:51.2232571Z, ParameterModified 2022-05-24T16:36:11.1705081Z, StructureModified 2022-05-24T16:36:11.1705081Z, UDAEnableTagReadback false
"9.TIMER_DELAY"
BEGIN
END_DATA_BLOCK

DATA_BLOCK "9.3.DLC_WA1"   // DB912
{ S7_Optimized_Access := 'TRUE' }
VERSION : 0.1
// stored: AutoNumber false, CodeModifiedDate 2026-01-15T16:25:51.1280002Z, CompileDate 2026-01-15T16:25:51.1337754Z, CreationDate 2026-01-15T16:22:49.8270549Z, DBAccessibleFromOPCUA true, DownloadWithoutReinit false, InstanceOfName 9.TIMER_DELAY, InstanceOfNumber 9, InstanceOfType FB, InterfaceModifiedDate 2022-05-24T16:36:11.1705081Z, IsConsistent true, IsKnowHowProtected false, IsRetainMemResEnabled false, MemoryReserve 100, ModifiedDate 2026-01-15T16:25:51.1280002Z, ParameterModified 2022-05-24T16:36:11.1705081Z, StructureModified 2022-05-24T16:36:11.1705081Z, UDAEnableTagReadback false
"9.TIMER_DELAY"
BEGIN
END_DATA_BLOCK

DATA_BLOCK "9.4.DLC_ADD1"   // DB914
{ S7_Optimized_Access := 'TRUE' }
VERSION : 0.1
// stored: AutoNumber false, CodeModifiedDate 2026-01-15T16:25:50.8619758Z, CompileDate 2026-01-15T16:25:50.8685917Z, CreationDate 2026-01-15T16:22:49.8270549Z, DBAccessibleFromOPCUA true, DownloadWithoutReinit false, InstanceOfName 9.TIMER_DELAY, InstanceOfNumber 9, InstanceOfType FB, InterfaceModifiedDate 2022-05-24T16:36:11.1705081Z, IsConsistent true, IsKnowHowProtected false, IsRetainMemResEnabled false, MemoryReserve 100, ModifiedDate 2026-01-15T16:25:50.8619758Z, ParameterModified 2022-05-24T16:36:11.1705081Z, StructureModified 2022-05-24T16:36:11.1705081Z, UDAEnableTagReadback false
"9.TIMER_DELAY"
BEGIN
END_DATA_BLOCK

DATA_BLOCK "9.4.DLC_ADD2"   // DB915
{ S7_Optimized_Access := 'TRUE' }
VERSION : 0.1
// stored: AutoNumber true, CodeModifiedDate 2026-01-15T16:25:55.9164676Z, CompileDate 2026-01-15T16:25:55.9210112Z, CreationDate 2026-01-15T16:22:49.8270549Z, DBAccessibleFromOPCUA true, DownloadWithoutReinit false, InstanceOfName 9.TIMER_DELAY, InstanceOfNumber 9, InstanceOfType FB, InterfaceModifiedDate 2022-05-24T16:36:11.1705081Z, IsConsistent true, IsKnowHowProtected false, IsRetainMemResEnabled false, MemoryReserve 100, ModifiedDate 2026-01-15T16:25:55.9164676Z, ParameterModified 2022-05-24T16:36:11.1705081Z, StructureModified 2022-05-24T16:36:11.1705081Z, UDAEnableTagReadback false
"9.TIMER_DELAY"
BEGIN
END_DATA_BLOCK

DATA_BLOCK "9.4.DLC_ADD3"   // DB916
{ S7_Optimized_Access := 'TRUE' }
VERSION : 0.1
// stored: AutoNumber true, CodeModifiedDate 2026-01-15T16:25:55.9010761Z, CompileDate 2026-01-15T16:25:55.9063674Z, CreationDate 2026-01-15T16:22:49.8270549Z, DBAccessibleFromOPCUA true, DownloadWithoutReinit false, InstanceOfName 9.TIMER_DELAY, InstanceOfNumber 9, InstanceOfType FB, InterfaceModifiedDate 2022-05-24T16:36:11.1705081Z, IsConsistent true, IsKnowHowProtected false, IsRetainMemResEnabled false, MemoryReserve 100, ModifiedDate 2026-01-15T16:25:55.9010761Z, ParameterModified 2022-05-24T16:36:11.1705081Z, StructureModified 2022-05-24T16:36:11.1705081Z, UDAEnableTagReadback false
"9.TIMER_DELAY"
BEGIN
END_DATA_BLOCK

DATA_BLOCK "9.4.DLC_ADD4"   // DB917
{ S7_Optimized_Access := 'TRUE' }
VERSION : 0.1
// stored: AutoNumber true, CodeModifiedDate 2026-01-15T16:25:55.8843515Z, CompileDate 2026-01-15T16:25:55.8884236Z, CreationDate 2026-01-15T16:22:49.8270549Z, DBAccessibleFromOPCUA true, DownloadWithoutReinit false, InstanceOfName 9.TIMER_DELAY, InstanceOfNumber 9, InstanceOfType FB, InterfaceModifiedDate 2022-05-24T16:36:11.1705081Z, IsConsistent true, IsKnowHowProtected false, IsRetainMemResEnabled false, MemoryReserve 100, ModifiedDate 2026-01-15T16:25:55.8843515Z, ParameterModified 2022-05-24T16:36:11.1705081Z, StructureModified 2022-05-24T16:36:11.1705081Z, UDAEnableTagReadback false
"9.TIMER_DELAY"
BEGIN
END_DATA_BLOCK

DATA_BLOCK "9.4.DLC_ADD5"   // DB918
{ S7_Optimized_Access := 'TRUE' }
VERSION : 0.1
// stored: AutoNumber true, CodeModifiedDate 2026-01-15T16:25:55.8681219Z, CompileDate 2026-01-15T16:25:55.8727468Z, CreationDate 2026-01-15T16:22:49.8270549Z, DBAccessibleFromOPCUA true, DownloadWithoutReinit false, InstanceOfName 9.TIMER_DELAY, InstanceOfNumber 9, InstanceOfType FB, InterfaceModifiedDate 2022-05-24T16:36:11.1705081Z, IsConsistent true, IsKnowHowProtected false, IsRetainMemResEnabled false, MemoryReserve 100, ModifiedDate 2026-01-15T16:25:55.8681219Z, ParameterModified 2022-05-24T16:36:11.1705081Z, StructureModified 2022-05-24T16:36:11.1705081Z, UDAEnableTagReadback false
"9.TIMER_DELAY"
BEGIN
END_DATA_BLOCK

DATA_BLOCK "9.4.DLC_ADD6"   // DB919
{ S7_Optimized_Access := 'TRUE' }
VERSION : 0.1
// stored: AutoNumber true, CodeModifiedDate 2026-01-15T16:25:55.8491634Z, CompileDate 2026-01-15T16:25:55.8531826Z, CreationDate 2026-01-15T16:22:49.8270549Z, DBAccessibleFromOPCUA true, DownloadWithoutReinit false, InstanceOfName 9.TIMER_DELAY, InstanceOfNumber 9, InstanceOfType FB, InterfaceModifiedDate 2022-05-24T16:36:11.1705081Z, IsConsistent true, IsKnowHowProtected false, IsRetainMemResEnabled false, MemoryReserve 100, ModifiedDate 2026-01-15T16:25:55.8491634Z, ParameterModified 2022-05-24T16:36:11.1705081Z, StructureModified 2022-05-24T16:36:11.1705081Z, UDAEnableTagReadback false
"9.TIMER_DELAY"
BEGIN
END_DATA_BLOCK

DATA_BLOCK "9.5.DLR_AGG1"   // DB920
{ S7_Optimized_Access := 'TRUE' }
VERSION : 0.1
// stored: AutoNumber false, CodeModifiedDate 2026-01-15T16:25:51.2934448Z, CompileDate 2026-01-15T16:25:51.2995118Z, CreationDate 2026-01-15T16:22:49.8270549Z, DBAccessibleFromOPCUA true, DownloadWithoutReinit false, InstanceOfName 9.TIMER_DELAY, InstanceOfNumber 9, InstanceOfType FB, InterfaceModifiedDate 2022-05-24T16:36:11.1705081Z, IsConsistent true, IsKnowHowProtected false, IsRetainMemResEnabled false, MemoryReserve 100, ModifiedDate 2026-01-15T16:25:51.2934448Z, ParameterModified 2022-05-24T16:36:11.1705081Z, StructureModified 2022-05-24T16:36:11.1705081Z, UDAEnableTagReadback false
"9.TIMER_DELAY"
BEGIN
END_DATA_BLOCK

DATA_BLOCK "9.5.DLR_IND_AGG1"   // DB20
{ S7_Optimized_Access := 'TRUE' }
VERSION : 0.1
// stored: AutoNumber true, CodeModifiedDate 2026-01-15T16:25:51.0342418Z, CompileDate 2026-01-15T16:25:51.0383137Z, CreationDate 2026-01-15T16:22:49.8270549Z, DBAccessibleFromOPCUA true, DownloadWithoutReinit false, InstanceOfName 9.TIMER_DELAY, InstanceOfNumber 9, InstanceOfType FB, InterfaceModifiedDate 2022-05-24T16:36:11.1705081Z, IsConsistent true, IsKnowHowProtected false, IsRetainMemResEnabled false, MemoryReserve 100, ModifiedDate 2026-01-15T16:25:51.0342418Z, ParameterModified 2022-05-24T16:36:11.1705081Z, StructureModified 2022-05-24T16:36:11.1705081Z, UDAEnableTagReadback false
"9.TIMER_DELAY"
BEGIN
END_DATA_BLOCK

DATA_BLOCK "9.5.DLR_IND_AGG2"   // DB24
{ S7_Optimized_Access := 'TRUE' }
VERSION : 0.1
// stored: AutoNumber true, CodeModifiedDate 2026-01-15T16:25:52.2021386Z, CompileDate 2026-01-15T16:25:52.2076549Z, CreationDate 2026-01-15T16:22:49.8270549Z, DBAccessibleFromOPCUA true, DownloadWithoutReinit false, InstanceOfName 9.TIMER_DELAY, InstanceOfNumber 9, InstanceOfType FB, InterfaceModifiedDate 2022-05-24T16:36:11.1705081Z, IsConsistent true, IsKnowHowProtected false, IsRetainMemResEnabled false, MemoryReserve 100, ModifiedDate 2026-01-15T16:25:52.2021386Z, ParameterModified 2022-05-24T16:36:11.1705081Z, StructureModified 2022-05-24T16:36:11.1705081Z, UDAEnableTagReadback false
"9.TIMER_DELAY"
BEGIN
END_DATA_BLOCK

DATA_BLOCK "9.5.DLR_IND_AGG3"   // DB28
{ S7_Optimized_Access := 'TRUE' }
VERSION : 0.1
// stored: AutoNumber true, CodeModifiedDate 2026-01-15T16:25:52.1579158Z, CompileDate 2026-01-15T16:25:52.1632354Z, CreationDate 2026-01-15T16:22:49.8270549Z, DBAccessibleFromOPCUA true, DownloadWithoutReinit false, InstanceOfName 9.TIMER_DELAY, InstanceOfNumber 9, InstanceOfType FB, InterfaceModifiedDate 2022-05-24T16:36:11.1705081Z, IsConsistent true, IsKnowHowProtected false, IsRetainMemResEnabled false, MemoryReserve 100, ModifiedDate 2026-01-15T16:25:52.1579158Z, ParameterModified 2022-05-24T16:36:11.1705081Z, StructureModified 2022-05-24T16:36:11.1705081Z, UDAEnableTagReadback false
"9.TIMER_DELAY"
BEGIN
END_DATA_BLOCK

DATA_BLOCK "9.5.DLR_IND_AGG4"   // DB30
{ S7_Optimized_Access := 'TRUE' }
VERSION : 0.1
// stored: AutoNumber true, CodeModifiedDate 2026-01-15T16:25:52.0241256Z, CompileDate 2026-01-15T16:25:52.0298162Z, CreationDate 2026-01-15T16:22:49.8270549Z, DBAccessibleFromOPCUA true, DownloadWithoutReinit false, InstanceOfName 9.TIMER_DELAY, InstanceOfNumber 9, InstanceOfType FB, InterfaceModifiedDate 2022-05-24T16:36:11.1705081Z, IsConsistent true, IsKnowHowProtected false, IsRetainMemResEnabled false, MemoryReserve 100, ModifiedDate 2026-01-15T16:25:52.0241256Z, ParameterModified 2022-05-24T16:36:11.1705081Z, StructureModified 2022-05-24T16:36:11.1705081Z, UDAEnableTagReadback false
"9.TIMER_DELAY"
BEGIN
END_DATA_BLOCK

DATA_BLOCK "9.5.DLR_IND_AGG5"   // DB34
{ S7_Optimized_Access := 'TRUE' }
VERSION : 0.1
// stored: AutoNumber true, CodeModifiedDate 2026-01-15T16:25:51.9127485Z, CompileDate 2026-01-15T16:25:51.9188212Z, CreationDate 2026-01-15T16:22:49.8270549Z, DBAccessibleFromOPCUA true, DownloadWithoutReinit false, InstanceOfName 9.TIMER_DELAY, InstanceOfNumber 9, InstanceOfType FB, InterfaceModifiedDate 2022-05-24T16:36:11.1705081Z, IsConsistent true, IsKnowHowProtected false, IsRetainMemResEnabled false, MemoryReserve 100, ModifiedDate 2026-01-15T16:25:51.9127485Z, ParameterModified 2022-05-24T16:36:11.1705081Z, StructureModified 2022-05-24T16:36:11.1705081Z, UDAEnableTagReadback false
"9.TIMER_DELAY"
BEGIN
END_DATA_BLOCK

DATA_BLOCK "9.6.DLR_CEM1"   // DB926
{ S7_Optimized_Access := 'TRUE' }
VERSION : 0.1
// stored: AutoNumber false, CodeModifiedDate 2026-01-15T16:25:51.2763773Z, CompileDate 2026-01-15T16:25:51.2831109Z, CreationDate 2026-01-15T16:22:49.8270549Z, DBAccessibleFromOPCUA true, DownloadWithoutReinit false, InstanceOfName 9.TIMER_DELAY, InstanceOfNumber 9, InstanceOfType FB, InterfaceModifiedDate 2022-05-24T16:36:11.1705081Z, IsConsistent true, IsKnowHowProtected false, IsRetainMemResEnabled false, MemoryReserve 100, ModifiedDate 2026-01-15T16:25:51.2763773Z, ParameterModified 2022-05-24T16:36:11.1705081Z, StructureModified 2022-05-24T16:36:11.1705081Z, UDAEnableTagReadback false
"9.TIMER_DELAY"
BEGIN
END_DATA_BLOCK

DATA_BLOCK "9.6.DLR_WAT1"   // DB928
{ S7_Optimized_Access := 'TRUE' }
VERSION : 0.1
// stored: AutoNumber false, CodeModifiedDate 2026-01-15T16:25:51.1685507Z, CompileDate 2026-01-15T16:25:51.174575Z, CreationDate 2026-01-15T16:22:49.8270549Z, DBAccessibleFromOPCUA true, DownloadWithoutReinit false, InstanceOfName 9.TIMER_DELAY, InstanceOfNumber 9, InstanceOfType FB, InterfaceModifiedDate 2022-05-24T16:36:11.1705081Z, IsConsistent true, IsKnowHowProtected false, IsRetainMemResEnabled false, MemoryReserve 100, ModifiedDate 2026-01-15T16:25:51.1685507Z, ParameterModified 2022-05-24T16:36:11.1705081Z, StructureModified 2022-05-24T16:36:11.1705081Z, UDAEnableTagReadback false
"9.TIMER_DELAY"
BEGIN
END_DATA_BLOCK

DATA_BLOCK "9.7.DLR_ADD1"   // DB930
{ S7_Optimized_Access := 'TRUE' }
VERSION : 0.1
// stored: AutoNumber false, CodeModifiedDate 2026-01-15T16:25:51.0908241Z, CompileDate 2026-01-15T16:25:51.0955047Z, CreationDate 2026-01-15T16:22:49.8270549Z, DBAccessibleFromOPCUA true, DownloadWithoutReinit false, InstanceOfName 9.TIMER_DELAY, InstanceOfNumber 9, InstanceOfType FB, InterfaceModifiedDate 2022-05-24T16:36:11.1705081Z, IsConsistent true, IsKnowHowProtected false, IsRetainMemResEnabled false, MemoryReserve 100, ModifiedDate 2026-01-15T16:25:51.0908241Z, ParameterModified 2022-05-24T16:36:11.1705081Z, StructureModified 2022-05-24T16:36:11.1705081Z, UDAEnableTagReadback false
"9.TIMER_DELAY"
BEGIN
END_DATA_BLOCK

DATA_BLOCK "9.8.DLXA_PTG 48"   // DB948
{ S7_Optimized_Access := 'TRUE' }
VERSION : 0.1
// stored: AutoNumber false, CodeModifiedDate 2026-01-15T16:25:55.8332274Z, CompileDate 2026-01-15T16:25:55.8384648Z, CreationDate 2026-01-15T16:22:49.8270549Z, DBAccessibleFromOPCUA true, DownloadWithoutReinit false, InstanceOfName 9.TIMER_DELAY, InstanceOfNumber 9, InstanceOfType FB, InterfaceModifiedDate 2022-05-24T16:36:11.1705081Z, IsConsistent true, IsKnowHowProtected false, IsRetainMemResEnabled false, MemoryReserve 100, ModifiedDate 2026-01-15T16:25:55.8332274Z, ParameterModified 2022-05-24T16:36:11.1705081Z, StructureModified 2022-05-24T16:36:11.1705081Z, UDAEnableTagReadback false
"9.TIMER_DELAY"
BEGIN
END_DATA_BLOCK

DATA_BLOCK "9.8.DLX_AGG1"   // DB947
{ S7_Optimized_Access := 'TRUE' }
VERSION : 0.1
// stored: AutoNumber false, CodeModifiedDate 2026-01-15T16:25:55.9955664Z, CompileDate 2026-01-15T16:25:56.0026563Z, CreationDate 2026-01-15T16:22:49.8270549Z, DBAccessibleFromOPCUA true, DownloadWithoutReinit false, InstanceOfName 9.TIMER_DELAY, InstanceOfNumber 9, InstanceOfType FB, InterfaceModifiedDate 2022-05-24T16:36:11.1705081Z, IsConsistent true, IsKnowHowProtected false, IsRetainMemResEnabled false, MemoryReserve 100, ModifiedDate 2026-01-15T16:25:55.9955664Z, ParameterModified 2022-05-24T16:36:11.1705081Z, StructureModified 2022-05-24T16:36:11.1705081Z, UDAEnableTagReadback false
"9.TIMER_DELAY"
BEGIN
END_DATA_BLOCK
